LIN {X 0,Y 262.981,Z 430.812,A -85,B 0,C 180,E1 -18278.581,E2 -18278.581} C_VEL
LIN {X 0,Y 263.836,Z 425.981,A -85,B 0,C 180,E1 -18280.746,E2 -18280.746} C_VEL
LIN {X 0,Y 264.818,Z 420.507,A -85,B 0,C 180,E1 -18282.646,E2 -18282.646} C_VEL
LIN {X 0,Y 266.141,Z 413.615,A -85,B 0,C 180,E1 -18284.528,E2 -18284.528} C_VEL
LIN {X 0,Y 267.438,Z 405.7,A -85,B 0,C 180,E1 -18286.212,E2 -18286.212} C_VEL
LIN {X 0,Y 268.494,Z 398.154,A -85,B 0,C 180,E1 -18287.518,E2 -18287.518} C_VEL
LIN {X 0,Y 269.51,Z 390.236,A -85,B 0,C 180,E1 -18288.628,E2 -18288.628} C_VEL
LIN {X 0,Y 270.479,Z 382.045,A -85,B 0,C 180,E1 -18289.544,E2 -18289.544} C_VEL
LIN {X 0,Y 271.262,Z 373.736,A -85,B 0,C 180,E1 -18290.274,E2 -18290.274} C_VEL
LIN {X 0,Y 271.665,Z 364.754,A -85,B 0,C 180,E1 -18290.886,E2 -18290.886} C_VEL
LIN {X 0,Y 272.024,Z 355.186,A -85,B 0,C 180,E1 -18291.32,E2 -18291.32} C_VEL
LIN {X 0,Y 273.127,Z 306.683,A -85,B 0,C 180,E1 -18292.613,E2 -18292.613} C_VEL
LIN {X 0,Y 268.619,Z 295.095,A -85,B 0,C 180,E1 -18293.353,E2 -18293.353} C_VEL
LIN {X 0,Y 263.217,Z 282.947,A -85,B 0,C 180,E1 -18294.227,E2 -18294.227} C_VEL
LIN {X 0,Y 263.154,Z 282.519,A -85,B 0,C 180,E1 -18294.298,E2 -18294.298} C_VEL
LIN {X 0,Y 263.116,Z 282.525,A -85,B 0,C 180,E1 -18298.736,E2 -18298.736} C_VEL
LIN {X 0,Y 263.124,Z 282.523,A -85,B 0,C 180,E1 -18302.288,E2 -18302.288} C_VEL
LIN {X 0,Y 263.151,Z 282.514,A -85,B 0,C 180,E1 -18305.983,E2 -18305.983} C_VEL
LIN {X 0,Y 263.069,Z 282.528,A -85,B 0,C 180,E1 -18309.878,E2 -18309.878} C_VEL
LIN {X 0,Y 263.073,Z 282.528,A -85,B 0,C 180,E1 -18313.993,E2 -18313.993} C_VEL
LIN {X 0,Y 263.071,Z 282.519,A -85,B 0,C 180,E1 -18318.096,E2 -18318.096} C_VEL
LIN {X 0,Y 263.099,Z 282.522,A -85,B 0,C 180,E1 -18322.093,E2 -18322.093} C_VEL
LIN {X 0,Y 263.148,Z 282.518,A -85,B 0,C 180,E1 -18325.885,E2 -18325.885} C_VEL
LIN {X 0,Y 263.106,Z 282.524,A -85,B 0,C 180,E1 -18329.501,E2 -18329.501} C_VEL
LIN {X 0,Y 263.125,Z 282.517,A -85,B 0,C 180,E1 -18332.995,E2 -18332.995} C_VEL
LIN {X 0,Y 263.139,Z 282.517,A -85,B 0,C 180,E1 -18336.383,E2 -18336.383} C_VEL
LIN {X 0,Y 263.204,Z 282.511,A -85,B 0,C 180,E1 -18339.688,E2 -18339.688} C_VEL
LIN {X 0,Y 263.283,Z 282.49,A -85,B 0,C 180,E1 -18344.518,E2 -18344.518} C_VEL
LIN {X 0,Y 263.327,Z 282.496,A -85,B 0,C 180,E1 -18349.232,E2 -18349.232} C_VEL
LIN {X 0,Y 263.521,Z 282.471,A -85,B 0,C 180,E1 -18352.337,E2 -18352.337} C_VEL
LIN {X 0,Y 263.728,Z 282.438,A -85,B 0,C 180,E1 -18358.473,E2 -18358.473} C_VEL
LIN {X 0,Y 263.728,Z 282.444,A -85,B 0,C 180,E1 -18361.527,E2 -18361.527} C_VEL
LIN {X 0,Y 263.51,Z 282.471,A -85,B 0,C 180,E1 -18363.027,E2 -18363.027} C_VEL
LIN {X 0,Y 262.791,Z 282.568,A -85,B 0,C 180,E1 -18364.302,E2 -18364.302} C_VEL
LIN {X 0,Y 259.971,Z 282.922,A -85,B 0,C 180,E1 -18366.382,E2 -18366.382} C_VEL
LIN {X 0,Y 256.734,Z 283.316,A -85,B 0,C 180,E1 -18368.941,E2 -18368.941} C_VEL
LIN {X 0,Y 256.351,Z 283.36,A -85,B 0,C 180,E1 -18369.826,E2 -18369.826} C_VEL
LIN {X 0,Y 256.196,Z 283.384,A -85,B 0,C 180,E1 -18374.293,E2 -18374.293} C_VEL
LIN {X 0,Y 256.142,Z 283.39,A -85,B 0,C 180,E1 -18377.567,E2 -18377.567} C_VEL
LIN {X 0,Y 256.114,Z 283.392,A -85,B 0,C 180,E1 -18381.097,E2 -18381.097} C_VEL
LIN {X 0,Y 256.077,Z 283.396,A -85,B 0,C 180,E1 -18385.087,E2 -18385.087} C_VEL
LIN {X 0,Y 256.071,Z 283.4,A -85,B 0,C 180,E1 -18388.57,E2 -18388.57} C_VEL
LIN {X 0,Y 256.065,Z 283.404,A -85,B 0,C 180,E1 -18391.7,E2 -18391.7} C_VEL
LIN {X 0,Y 256.074,Z 283.402,A -85,B 0,C 180,E1 -18395.194,E2 -18395.194} C_VEL
LIN {X 0,Y 256.041,Z 283.407,A -85,B 0,C 180,E1 -18399.147,E2 -18399.147} C_VEL
LIN {X 0,Y 256.018,Z 283.41,A -85,B 0,C 180,E1 -18403.336,E2 -18403.336} C_VEL
LIN {X 0,Y 256.029,Z 283.405,A -85,B 0,C 180,E1 -18407.829,E2 -18407.829} C_VEL
LIN {X 0,Y 256.063,Z 283.403,A -85,B 0,C 180,E1 -18410.858,E2 -18410.858} C_VEL
LIN {X 0,Y 256.122,Z 283.395,A -85,B 0,C 180,E1 -18412.867,E2 -18412.867} C_VEL
LIN {X 0,Y 256.173,Z 283.581,A -85,B 0,C 180,E1 -18416.931,E2 -18416.931} C_VEL
LIN {X 0,Y 258.108,Z 292.95,A -85,B 0,C 180,E1 -18420.653,E2 -18420.653} C_VEL
LIN {X 0,Y 259.582,Z 301.431,A -85,B 0,C 180,E1 -18423.857,E2 -18423.857} C_VEL
LIN {X 0,Y 259.06,Z 305.592,A -85,B 0,C 180,E1 -18425.289,E2 -18425.289} C_VEL
LIN {X 0,Y 262.798,Z 329.088,A -85,B 0,C 180,E1 -18426.351,E2 -18426.351} C_VEL
LIN {X 0,Y 265.475,Z 352.015,A -85,B 0,C 180,E1 -18427.258,E2 -18427.258} C_VEL
LIN {X 0,Y 264.769,Z 384.627,A -85,B 0,C 180,E1 -18428.186,E2 -18428.186} C_VEL
LIN {X 0,Y 263.962,Z 395.927,A -85,B 0,C 180,E1 -18428.742,E2 -18428.742} C_VEL
LIN {X 0,Y 262.729,Z 407.426,A -85,B 0,C 180,E1 -18429.651,E2 -18429.651} C_VEL
LIN {X 0,Y 261.591,Z 416.12,A -85,B 0,C 180,E1 -18430.582,E2 -18430.582} C_VEL
LIN {X 0,Y 260.318,Z 424.431,A -85,B 0,C 180,E1 -18431.71,E2 -18431.71} C_VEL
LIN {X 0,Y 259.057,Z 432.309,A -85,B 0,C 180,E1 -18433.045,E2 -18433.045} C_VEL
LIN {X 0,Y 257.772,Z 439.681,A -85,B 0,C 180,E1 -18434.585,E2 -18434.585} C_VEL
LIN {X 0,Y 256.42,Z 447.167,A -85,B 0,C 180,E1 -18436.529,E2 -18436.529} C_VEL
LIN {X 0,Y 255.25,Z 454.012,A -85,B 0,C 180,E1 -18438.888,E2 -18438.888} C_VEL
LIN {X 0,Y 254.567,Z 459.229,A -85,B 0,C 180,E1 -18441.267,E2 -18441.267} C_VEL
LIN {X 0,Y 254.177,Z 463.065,A -85,B 0,C 180,E1 -18443.651,E2 -18443.651} C_VEL
LIN {X 0,Y 254.081,Z 464.833,A -85,B 0,C 180,E1 -18445.241,E2 -18445.241} C_VEL
LIN {X 0,Y 254.147,Z 466.105,A -85,B 0,C 180,E1 -18446.83,E2 -18446.83} C_VEL
LIN {X 0,Y 254.188,Z 466.894,A -85,B 0,C 180,E1 -18448.416,E2 -18448.416} C_VEL
LIN {X 0,Y 254.272,Z 467.194,A -85,B 0,C 180,E1 -18450.001,E2 -18450.001} C_VEL
LIN {X 0,Y 254.188,Z 466.886,A -85,B 0,C 180,E1 -18451.585,E2 -18451.585} C_VEL
LIN {X 0,Y 254.148,Z 466.082,A -85,B 0,C 180,E1 -18453.171,E2 -18453.171} C_VEL
LIN {X 0,Y 254.159,Z 464.076,A -85,B 0,C 180,E1 -18455.456,E2 -18455.456} C_VEL
LIN {X 0,Y 254.389,Z 460.655,A -85,B 0,C 180,E1 -18457.941,E2 -18457.941} C_VEL
LIN {X 0,Y 254.981,Z 455.856,A -85,B 0,C 180,E1 -18460.322,E2 -18460.322} C_VEL
LIN {X 0,Y 255.815,Z 450.672,A -85,B 0,C 180,E1 -18462.294,E2 -18462.294} C_VEL
LIN {X 0,Y 256.654,Z 445.61,A -85,B 0,C 180,E1 -18463.864,E2 -18463.864} C_VEL
LIN {X 0,Y 257.74,Z 439.523,A -85,B 0,C 180,E1 -18465.419,E2 -18465.419} C_VEL
LIN {X 0,Y 259.06,Z 432.125,A -85,B 0,C 180,E1 -18466.957,E2 -18466.957} C_VEL
LIN {X 0,Y 260.36,Z 424.206,A -85,B 0,C 180,E1 -18468.289,E2 -18468.289} C_VEL
LIN {X 0,Y 261.578,Z 415.838,A -85,B 0,C 180,E1 -18469.421,E2 -18469.421} C_VEL
LIN {X 0,Y 263.007,Z 404.764,A -85,B 0,C 180,E1 -18470.568,E2 -18470.568} C_VEL
LIN {X 0,Y 264.001,Z 394.383,A -85,B 0,C 180,E1 -18471.314,E2 -18471.314} C_VEL
LIN {X 0,Y 264.739,Z 384.752,A -85,B 0,C 180,E1 -18471.775,E2 -18471.775} C_VEL
LIN {X 0,Y 265.445,Z 352.252,A -85,B 0,C 180,E1 -18472.7,E2 -18472.7} C_VEL
LIN {X 0,Y 262.541,Z 327.679,A -85,B 0,C 180,E1 -18473.675,E2 -18473.675} C_VEL
LIN {X 0,Y 259.343,Z 307.499,A -85,B 0,C 180,E1 -18474.578,E2 -18474.578} C_VEL
LIN {X 0,Y 259.035,Z 305.586,A -85,B 0,C 180,E1 -18474.676,E2 -18474.676} C_VEL
LIN {X 0,Y 259.551,Z 301.335,A -85,B 0,C 180,E1 -18476.141,E2 -18476.141} C_VEL
LIN {X 0,Y 258.078,Z 292.765,A -85,B 0,C 180,E1 -18479.376,E2 -18479.376} C_VEL
LIN {X 0,Y 256.134,Z 283.389,A -85,B 0,C 180,E1 -18483.141,E2 -18483.141} C_VEL
LIN {X 0,Y 256.111,Z 283.397,A -85,B 0,C 180,E1 -18487.27,E2 -18487.27} C_VEL
LIN {X 0,Y 256.019,Z 283.409,A -85,B 0,C 180,E1 -18491.211,E2 -18491.211} C_VEL
LIN {X 0,Y 256.018,Z 283.407,A -85,B 0,C 180,E1 -18495.54,E2 -18495.54} C_VEL
LIN {X 0,Y 256.01,Z 283.411,A -85,B 0,C 180,E1 -18498.788,E2 -18498.788} C_VEL
LIN {X 0,Y 256.1,Z 283.399,A -85,B 0,C 180,E1 -18502.862,E2 -18502.862} C_VEL
LIN {X 0,Y 256.067,Z 283.402,A -85,B 0,C 180,E1 -18506.707,E2 -18506.707} C_VEL
LIN {X 0,Y 256.042,Z 283.406,A -85,B 0,C 180,E1 -18510.391,E2 -18510.391} C_VEL
LIN {X 0,Y 256.067,Z 283.402,A -85,B 0,C 180,E1 -18513.951,E2 -18513.951} C_VEL
LIN {X 0,Y 256.058,Z 283.401,A -85,B 0,C 180,E1 -18517.403,E2 -18517.403} C_VEL
LIN {X 0,Y 256.101,Z 283.395,A -85,B 0,C 180,E1 -18520.773,E2 -18520.773} C_VEL
LIN {X 0,Y 256.214,Z 283.382,A -85,B 0,C 180,E1 -18524.08,E2 -18524.08} C_VEL
LIN {X 0,Y 256.272,Z 283.37,A -85,B 0,C 180,E1 -18528.933,E2 -18528.933} C_VEL
LIN {X 0,Y 256.458,Z 283.334,A -85,B 0,C 180,E1 -18532.125,E2 -18532.125} C_VEL
LIN {X 0,Y 256.445,Z 283.351,A -85,B 0,C 180,E1 -18536.858,E2 -18536.858} C_VEL
LIN {X 0,Y 256.695,Z 283.32,A -85,B 0,C 180,E1 -18538.431,E2 -18538.431} C_VEL
LIN {X 0,Y 256.697,Z 283.312,A -85,B 0,C 180,E1 -18541.569,E2 -18541.569} C_VEL
LIN {X 0,Y 256.444,Z 283.345,A -85,B 0,C 180,E1 -18546.573,E2 -18546.573} C_VEL
LIN {X 0,Y 256.405,Z 283.359,A -85,B 0,C 180,E1 -18549.466,E2 -18549.466} C_VEL
LIN {X 0,Y 256.208,Z 283.369,A -85,B 0,C 180,E1 -18554.293,E2 -18554.293} C_VEL
LIN {X 0,Y 256.149,Z 283.385,A -85,B 0,C 180,E1 -18557.566,E2 -18557.566} C_VEL
LIN {X 0,Y 256.121,Z 283.393,A -85,B 0,C 180,E1 -18561.097,E2 -18561.097} C_VEL
LIN {X 0,Y 256.085,Z 283.398,A -85,B 0,C 180,E1 -18565.087,E2 -18565.087} C_VEL
LIN {X 0,Y 256.079,Z 283.397,A -85,B 0,C 180,E1 -18568.57,E2 -18568.57} C_VEL
LIN {X 0,Y 256.072,Z 283.397,A -85,B 0,C 180,E1 -18571.699,E2 -18571.699} C_VEL
LIN {X 0,Y 256.08,Z 283.388,A -85,B 0,C 180,E1 -18575.193,E2 -18575.193} C_VEL
LIN {X 0,Y 256.044,Z 283.403,A -85,B 0,C 180,E1 -18579.147,E2 -18579.147} C_VEL
LIN {X 0,Y 256.023,Z 283.399,A -85,B 0,C 180,E1 -18583.335,E2 -18583.335} C_VEL
LIN {X 0,Y 256.036,Z 283.404,A -85,B 0,C 180,E1 -18587.828,E2 -18587.828} C_VEL
LIN {X 0,Y 256.067,Z 283.378,A -85,B 0,C 180,E1 -18590.856,E2 -18590.856} C_VEL
LIN {X 0,Y 256.081,Z 283.395,A -85,B 0,C 180,E1 -18594.806,E2 -18594.806} C_VEL
LIN {X 0,Y 256.079,Z 283.398,A -85,B 0,C 180,E1 -18598.57,E2 -18598.57} C_VEL
LIN {X 0,Y 256.081,Z 283.399,A -85,B 0,C 180,E1 -18602.188,E2 -18602.188} C_VEL
LIN {X 0,Y 256.164,Z 283.505,A -85,B 0,C 180,E1 -18605.198,E2 -18605.198} C_VEL
LIN {X 0,Y 257.229,Z 286.37,A -85,B 0,C 180,E1 -18605.397,E2 -18605.397} C_VEL
LIN {X 0,Y 264.851,Z 303.493,A -85,B 0,C 180,E1 -18606.662,E2 -18606.662} C_VEL
LIN {X 0,Y 266.558,Z 308.226,A -85,B 0,C 180,E1 -18606.959,E2 -18606.959} C_VEL
LIN {X 0,Y 265.305,Z 356.614,A -85,B 0,C 180,E1 -18608.281,E2 -18608.281} C_VEL
LIN {X 0,Y 264.934,Z 366.352,A -85,B 0,C 180,E1 -18608.76,E2 -18608.76} C_VEL
LIN {X 0,Y 264.292,Z 377.392,A -85,B 0,C 180,E1 -18609.572,E2 -18609.572} C_VEL
LIN {X 0,Y 263.081,Z 388.176,A -85,B 0,C 180,E1 -18610.695,E2 -18610.695} C_VEL
LIN {X 0,Y 262.117,Z 395.319,A -85,B 0,C 180,E1 -18611.636,E2 -18611.636} C_VEL
LIN {X 0,Y 260.971,Z 403.419,A -85,B 0,C 180,E1 -18612.97,E2 -18612.97} C_VEL
LIN {X 0,Y 259.915,Z 410.098,A -85,B 0,C 180,E1 -18614.311,E2 -18614.311} C_VEL
LIN {X 0,Y 258.791,Z 416.422,A -85,B 0,C 180,E1 -18615.852,E2 -18615.852} C_VEL
LIN {X 0,Y 257.743,Z 421.68,A -85,B 0,C 180,E1 -18617.399,E2 -18617.399} C_VEL
LIN {X 0,Y 256.886,Z 426.065,A -85,B 0,C 180,E1 -18618.958,E2 -18618.958} C_VEL
LIN {X 0,Y 256.235,Z 429.71,A -85,B 0,C 180,E1 -18620.527,E2 -18620.527} C_VEL
LIN {X 0,Y 255.713,Z 432.686,A -85,B 0,C 180,E1 -18622.101,E2 -18622.101} C_VEL
LIN {X 0,Y 255.241,Z 434.992,A -85,B 0,C 180,E1 -18623.676,E2 -18623.676} C_VEL
LIN {X 0,Y 254.819,Z 436.748,A -85,B 0,C 180,E1 -18625.253,E2 -18625.253} C_VEL
LIN {X 0,Y 254.53,Z 438.013,A -85,B 0,C 180,E1 -18626.834,E2 -18626.834} C_VEL
LIN {X 0,Y 254.358,Z 438.81,A -85,B 0,C 180,E1 -18628.416,E2 -18628.416} C_VEL
LIN {X 0,Y 254.305,Z 439.113,A -85,B 0,C 180,E1 -18629.999,E2 -18629.999} C_VEL
LIN {X 0,Y 254.355,Z 438.836,A -85,B 0,C 180,E1 -18631.582,E2 -18631.582} C_VEL
LIN {X 0,Y 254.518,Z 438.09,A -85,B 0,C 180,E1 -18633.165,E2 -18633.165} C_VEL
LIN {X 0,Y 254.813,Z 436.878,A -85,B 0,C 180,E1 -18634.745,E2 -18634.745} C_VEL
LIN {X 0,Y 255.443,Z 434.037,A -85,B 0,C 180,E1 -18637.111,E2 -18637.111} C_VEL
LIN {X 0,Y 255.943,Z 431.454,A -85,B 0,C 180,E1 -18638.685,E2 -18638.685} C_VEL
LIN {X 0,Y 256.878,Z 426.37,A -85,B 0,C 180,E1 -18641.04,E2 -18641.04} C_VEL
LIN {X 0,Y 257.918,Z 420.896,A -85,B 0,C 180,E1 -18642.99,E2 -18642.99} C_VEL
LIN {X 0,Y 259.284,Z 414.003,A -85,B 0,C 180,E1 -18644.921,E2 -18644.921} C_VEL
LIN {X 0,Y 260.646,Z 406.088,A -85,B 0,C 180,E1 -18646.647,E2 -18646.647} C_VEL
LIN {X 0,Y 261.751,Z 398.541,A -85,B 0,C 180,E1 -18647.984,E2 -18647.984} C_VEL
LIN {X 0,Y 262.817,Z 390.621,A -85,B 0,C 180,E1 -18649.121,E2 -18649.121} C_VEL
LIN {X 0,Y 263.835,Z 382.429,A -85,B 0,C 180,E1 -18650.057,E2 -18650.057} C_VEL
LIN {X 0,Y 264.639,Z 374.119,A -85,B 0,C 180,E1 -18650.805,E2 -18650.805} C_VEL
LIN {X 0,Y 265.066,Z 365.134,A -85,B 0,C 180,E1 -18651.431,E2 -18651.431} C_VEL
LIN {X 0,Y 265.444,Z 355.6,A -85,B 0,C 180,E1 -18651.874,E2 -18651.874} C_VEL
LIN {X 0,Y 266.661,Z 308.565,A -85,B 0,C 180,E1 -18653.15,E2 -18653.15} C_VEL
LIN {X 0,Y 262.754,Z 298.437,A -85,B 0,C 180,E1 -18653.818,E2 -18653.818} C_VEL
LIN {X 0,Y 256.205,Z 284.082,A -85,B 0,C 180,E1 -18654.912,E2 -18654.912} C_VEL
LIN {X 0,Y 256.092,Z 283.403,A -85,B 0,C 180,E1 -18654.995,E2 -18654.995} C_VEL
LIN {X 0,Y 256.074,Z 283.402,A -85,B 0,C 180,E1 -18658.568,E2 -18658.568} C_VEL
LIN {X 0,Y 256.068,Z 283.4,A -85,B 0,C 180,E1 -18661.698,E2 -18661.698} C_VEL
LIN {X 0,Y 256.076,Z 283.396,A -85,B 0,C 180,E1 -18665.193,E2 -18665.193} C_VEL
LIN {X 0,Y 256.039,Z 283.403,A -85,B 0,C 180,E1 -18669.147,E2 -18669.147} C_VEL
LIN {X 0,Y 256.018,Z 283.403,A -85,B 0,C 180,E1 -18673.335,E2 -18673.335} C_VEL
LIN {X 0,Y 256.026,Z 283.395,A -85,B 0,C 180,E1 -18677.829,E2 -18677.829} C_VEL
LIN {X 0,Y 256.038,Z 283.4,A -85,B 0,C 180,E1 -18680.852,E2 -18680.852} C_VEL
LIN {X 0,Y 256.074,Z 283.396,A -85,B 0,C 180,E1 -18684.806,E2 -18684.806} C_VEL
LIN {X 0,Y 256.074,Z 283.396,A -85,B 0,C 180,E1 -18688.57,E2 -18688.57} C_VEL
LIN {X 0,Y 256.082,Z 283.393,A -85,B 0,C 180,E1 -18692.189,E2 -18692.189} C_VEL
LIN {X 0,Y 256.128,Z 283.392,A -85,B 0,C 180,E1 -18695.695,E2 -18695.695} C_VEL
LIN {X 0,Y 256.119,Z 283.394,A -85,B 0,C 180,E1 -18699.101,E2 -18699.101} C_VEL
LIN {X 0,Y 256.208,Z 283.37,A -85,B 0,C 180,E1 -18704.079,E2 -18704.079} C_VEL
LIN {X 0,Y 256.271,Z 283.374,A -85,B 0,C 180,E1 -18708.932,E2 -18708.932} C_VEL
LIN {X 0,Y 256.463,Z 283.349,A -85,B 0,C 180,E1 -18712.125,E2 -18712.125} C_VEL
LIN {X 0,Y 256.443,Z 283.338,A -85,B 0,C 180,E1 -18716.858,E2 -18716.858} C_VEL
LIN {X 0,Y 256.69,Z 283.313,A -85,B 0,C 180,E1 -18718.431,E2 -18718.431} C_VEL
LIN {X 0,Y 256.69,Z 283.321,A -85,B 0,C 180,E1 -18721.569,E2 -18721.569} C_VEL
LIN {X 0,Y 256.448,Z 283.352,A -85,B 0,C 180,E1 -18726.293,E2 -18726.293} C_VEL
LIN {X 0,Y 256.397,Z 283.356,A -85,B 0,C 180,E1 -18729.466,E2 -18729.466} C_VEL
LIN {X 0,Y 256.351,Z 283.36,A -85,B 0,C 180,E1 -18729.826,E2 -18729.826} C_VEL
LIN {X 0,Y 255.59,Z 283.457,A -85,B 0,C 180,E1 -18731.135,E2 -18731.135} C_VEL
LIN {X 0,Y 252.714,Z 283.817,A -85,B 0,C 180,E1 -18733.27,E2 -18733.27} C_VEL
LIN {X 0,Y 250.299,Z 284.12,A -85,B 0,C 180,E1 -18735.006,E2 -18735.006} C_VEL
LIN {X 0,Y 249.225,Z 284.253,A -85,B 0,C 180,E1 -18736.352,E2 -18736.352} C_VEL
LIN {X 0,Y 249.113,Z 284.265,A -85,B 0,C 180,E1 -18736.809,E2 -18736.809} C_VEL
LIN {X 0,Y 249.038,Z 284.275,A -85,B 0,C 180,E1 -18741.522,E2 -18741.522} C_VEL
LIN {X 0,Y 249.038,Z 284.275,A -85,B 0,C 180,E1 -18745.44,E2 -18745.44} C_VEL
LIN {X 0,Y 249.019,Z 284.279,A -85,B 0,C 180,E1 -18748.968,E2 -18748.968} C_VEL
LIN {X 0,Y 249.021,Z 284.279,A -85,B 0,C 180,E1 -18752.427,E2 -18752.427} C_VEL
LIN {X 0,Y 249.006,Z 284.281,A -85,B 0,C 180,E1 -18756.349,E2 -18756.349} C_VEL
LIN {X 0,Y 248.971,Z 284.285,A -85,B 0,C 180,E1 -18760.485,E2 -18760.485} C_VEL
LIN {X 0,Y 248.958,Z 284.289,A -85,B 0,C 180,E1 -18764.889,E2 -18764.889} C_VEL
LIN {X 0,Y 248.975,Z 284.287,A -85,B 0,C 180,E1 -18767.355,E2 -18767.355} C_VEL
LIN {X 0,Y 249.037,Z 284.276,A -85,B 0,C 180,E1 -18772.202,E2 -18772.202} C_VEL
LIN {X 0,Y 249.076,Z 284.43,A -85,B 0,C 180,E1 -18776.378,E2 -18776.378} C_VEL
LIN {X 0,Y 251.064,Z 293.716,A -85,B 0,C 180,E1 -18780.201,E2 -18780.201} C_VEL
LIN {X 0,Y 252.606,Z 302.339,A -85,B 0,C 180,E1 -18783.568,E2 -18783.568} C_VEL
LIN {X 0,Y 252.335,Z 305.187,A -85,B 0,C 180,E1 -18784.586,E2 -18784.586} C_VEL
LIN {X 0,Y 256.291,Z 330.056,A -85,B 0,C 180,E1 -18785.753,E2 -18785.753} C_VEL
LIN {X 0,Y 258.774,Z 351.122,A -85,B 0,C 180,E1 -18786.62,E2 -18786.62} C_VEL
LIN {X 0,Y 258.889,Z 358.477,A -85,B 0,C 180,E1 -18786.847,E2 -18786.847} C_VEL
LIN {X 0,Y 258.164,Z 384.249,A -85,B 0,C 180,E1 -18787.598,E2 -18787.598} C_VEL
LIN {X 0,Y 257.321,Z 396.001,A -85,B 0,C 180,E1 -18788.198,E2 -18788.198} C_VEL
LIN {X 0,Y 256.091,Z 407.04,A -85,B 0,C 180,E1 -18789.099,E2 -18789.099} C_VEL
LIN {X 0,Y 254.911,Z 415.733,A -85,B 0,C 180,E1 -18790.052,E2 -18790.052} C_VEL
LIN {X 0,Y 253.575,Z 424.042,A -85,B 0,C 180,E1 -18791.205,E2 -18791.205} C_VEL
LIN {X 0,Y 252.252,Z 431.919,A -85,B 0,C 180,E1 -18792.573,E2 -18792.573} C_VEL
LIN {X 0,Y 250.896,Z 439.29,A -85,B 0,C 180,E1 -18794.151,E2 -18794.151} C_VEL
LIN {X 0,Y 249.505,Z 446.776,A -85,B 0,C 180,E1 -18796.148,E2 -18796.148} C_VEL
LIN {X 0,Y 248.261,Z 453.62,A -85,B 0,C 180,E1 -18798.571,E2 -18798.571} C_VEL
LIN {X 0,Y 247.528,Z 458.837,A -85,B 0,C 180,E1 -18801.017,E2 -18801.017} C_VEL
LIN {X 0,Y 247.095,Z 462.673,A -85,B 0,C 180,E1 -18803.468,E2 -18803.468} C_VEL
LIN {X 0,Y 247.009,Z 464.442,A -85,B 0,C 180,E1 -18805.104,E2 -18805.104} C_VEL
LIN {X 0,Y 247.056,Z 465.713,A -85,B 0,C 180,E1 -18806.739,E2 -18806.739} C_VEL
LIN {X 0,Y 247.112,Z 466.503,A -85,B 0,C 180,E1 -18808.371,E2 -18808.371} C_VEL
LIN {X 0,Y 247.191,Z 466.803,A -85,B 0,C 180,E1 -18810.001,E2 -18810.001} C_VEL
LIN {X 0,Y 247.112,Z 466.495,A -85,B 0,C 180,E1 -18811.631,E2 -18811.631} C_VEL
LIN {X 0,Y 247.058,Z 465.69,A -85,B 0,C 180,E1 -18813.262,E2 -18813.262} C_VEL
LIN {X 0,Y 247.048,Z 463.966,A -85,B 0,C 180,E1 -18815.332,E2 -18815.332} C_VEL
LIN {X 0,Y 247.199,Z 461.449,A -85,B 0,C 180,E1 -18817.351,E2 -18817.351} C_VEL
LIN {X 0,Y 247.528,Z 458.765,A -85,B 0,C 180,E1 -18818.985,E2 -18818.985} C_VEL
LIN {X 0,Y 248.261,Z 453.526,A -85,B 0,C 180,E1 -18821.43,E2 -18821.43} C_VEL
LIN {X 0,Y 249.501,Z 446.639,A -85,B 0,C 180,E1 -18823.854,E2 -18823.854} C_VEL
LIN {X 0,Y 250.874,Z 439.127,A -85,B 0,C 180,E1 -18825.852,E2 -18825.852} C_VEL
LIN {X 0,Y 252.256,Z 431.729,A -85,B 0,C 180,E1 -18827.428,E2 -18827.428} C_VEL
LIN {X 0,Y 253.625,Z 423.81,A -85,B 0,C 180,E1 -18828.793,E2 -18828.793} C_VEL
LIN {X 0,Y 254.897,Z 415.441,A -85,B 0,C 180,E1 -18829.951,E2 -18829.951} C_VEL
LIN {X 0,Y 256.378,Z 404.365,A -85,B 0,C 180,E1 -18831.125,E2 -18831.125} C_VEL
LIN {X 0,Y 257.451,Z 393.688,A -85,B 0,C 180,E1 -18831.902,E2 -18831.902} C_VEL
LIN {X 0,Y 258.141,Z 384.504,A -85,B 0,C 180,E1 -18832.355,E2 -18832.355} C_VEL
LIN {X 0,Y 258.876,Z 352.874,A -85,B 0,C 180,E1 -18833.279,E2 -18833.279} C_VEL
LIN {X 0,Y 256.108,Z 329.071,A -85,B 0,C 180,E1 -18834.254,E2 -18834.254} C_VEL
LIN {X 0,Y 252.722,Z 307.666,A -85,B 0,C 180,E1 -18835.248,E2 -18835.248} C_VEL
LIN {X 0,Y 252.309,Z 305.175,A -85,B 0,C 180,E1 -18835.38,E2 -18835.38} C_VEL
LIN {X 0,Y 252.582,Z 302.221,A -85,B 0,C 180,E1 -18836.437,E2 -18836.437} C_VEL
LIN {X 0,Y 250.837,Z 292.374,A -85,B 0,C 180,E1 -18840.288,E2 -18840.288} C_VEL
LIN {X 0,Y 249.058,Z 284.27,A -85,B 0,C 180,E1 -18843.688,E2 -18843.688} C_VEL
LIN {X 0,Y 249.023,Z 284.278,A -85,B 0,C 180,E1 -18848.382,E2 -18848.382} C_VEL
LIN {X 0,Y 248.971,Z 284.287,A -85,B 0,C 180,E1 -18852.783,E2 -18852.783} C_VEL
LIN {X 0,Y 248.978,Z 284.285,A -85,B 0,C 180,E1 -18857.355,E2 -18857.355} C_VEL
LIN {X 0,Y 249.022,Z 284.28,A -85,B 0,C 180,E1 -18862.208,E2 -18862.208} C_VEL
LIN {X 0,Y 249.044,Z 284.275,A -85,B 0,C 180,E1 -18865.64,E2 -18865.64} C_VEL
LIN {X 0,Y 248.995,Z 284.281,A -85,B 0,C 180,E1 -18869.466,E2 -18869.466} C_VEL
LIN {X 0,Y 249.014,Z 284.278,A -85,B 0,C 180,E1 -18873.156,E2 -18873.156} C_VEL
LIN {X 0,Y 249.007,Z 284.28,A -85,B 0,C 180,E1 -18876.726,E2 -18876.726} C_VEL
LIN {X 0,Y 249.04,Z 284.276,A -85,B 0,C 180,E1 -18880.206,E2 -18880.206} C_VEL
LIN {X 0,Y 249.16,Z 284.261,A -85,B 0,C 180,E1 -18883.617,E2 -18883.617} C_VEL
LIN {X 0,Y 249.217,Z 284.249,A -85,B 0,C 180,E1 -18888.615,E2 -18888.615} C_VEL
LIN {X 0,Y 249.405,Z 284.211,A -85,B 0,C 180,E1 -18891.901,E2 -18891.901} C_VEL
LIN {X 0,Y 249.256,Z 284.242,A -85,B 0,C 180,E1 -18895.148,E2 -18895.148} C_VEL
LIN {X 0,Y 249.656,Z 284.197,A -85,B 0,C 180,E1 -18898.387,E2 -18898.387} C_VEL
LIN {X 0,Y 249.658,Z 284.187,A -85,B 0,C 180,E1 -18901.613,E2 -18901.613} C_VEL
LIN {X 0,Y 249.422,Z 284.22,A -85,B 0,C 180,E1 -18906.55,E2 -18906.55} C_VEL
LIN {X 0,Y 249.335,Z 284.238,A -85,B 0,C 180,E1 -18909.737,E2 -18909.737} C_VEL
LIN {X 0,Y 249.151,Z 284.245,A -85,B 0,C 180,E1 -18914.707,E2 -18914.707} C_VEL
LIN {X 0,Y 249.081,Z 284.265,A -85,B 0,C 180,E1 -18918.082,E2 -18918.082} C_VEL
LIN {X 0,Y 249.045,Z 284.273,A -85,B 0,C 180,E1 -18921.522,E2 -18921.522} C_VEL
LIN {X 0,Y 249.046,Z 284.274,A -85,B 0,C 180,E1 -18925.439,E2 -18925.439} C_VEL
LIN {X 0,Y 249.027,Z 284.277,A -85,B 0,C 180,E1 -18928.968,E2 -18928.968} C_VEL
LIN {X 0,Y 249.028,Z 284.274,A -85,B 0,C 180,E1 -18932.426,E2 -18932.426} C_VEL
LIN {X 0,Y 249.013,Z 284.272,A -85,B 0,C 180,E1 -18936.349,E2 -18936.349} C_VEL
LIN {X 0,Y 248.974,Z 284.282,A -85,B 0,C 180,E1 -18940.485,E2 -18940.485} C_VEL
LIN {X 0,Y 248.964,Z 284.286,A -85,B 0,C 180,E1 -18944.888,E2 -18944.888} C_VEL
LIN {X 0,Y 248.981,Z 284.284,A -85,B 0,C 180,E1 -18947.355,E2 -18947.355} C_VEL
LIN {X 0,Y 249.045,Z 284.247,A -85,B 0,C 180,E1 -18952.2,E2 -18952.2} C_VEL
LIN {X 0,Y 249.045,Z 284.274,A -85,B 0,C 180,E1 -18955.639,E2 -18955.639} C_VEL
LIN {X 0,Y 248.996,Z 284.282,A -85,B 0,C 180,E1 -18959.465,E2 -18959.465} C_VEL
LIN {X 0,Y 249.025,Z 284.28,A -85,B 0,C 180,E1 -18963.156,E2 -18963.156} C_VEL
LIN {X 0,Y 249.096,Z 284.45,A -85,B 0,C 180,E1 -18964.46,E2 -18964.46} C_VEL
LIN {X 0,Y 250.147,Z 287.197,A -85,B 0,C 180,E1 -18964.663,E2 -18964.663} C_VEL
LIN {X 0,Y 258.118,Z 304.653,A -85,B 0,C 180,E1 -18966.037,E2 -18966.037} C_VEL
LIN {X 0,Y 260.08,Z 310.304,A -85,B 0,C 180,E1 -18966.4,E2 -18966.4} C_VEL
LIN {X 0,Y 258.783,Z 355.728,A -85,B 0,C 180,E1 -18967.653,E2 -18967.653} C_VEL
LIN {X 0,Y 258.446,Z 365.095,A -85,B 0,C 180,E1 -18968.095,E2 -18968.095} C_VEL
LIN {X 0,Y 257.918,Z 374.201,A -85,B 0,C 180,E1 -18968.73,E2 -18968.73} C_VEL
LIN {X 0,Y 257.038,Z 383.51,A -85,B 0,C 180,E1 -18969.597,E2 -18969.597} C_VEL
LIN {X 0,Y 255.718,Z 393.062,A -85,B 0,C 180,E1 -18970.743,E2 -18970.743} C_VEL
LIN {X 0,Y 254.369,Z 402.799,A -85,B 0,C 180,E1 -18972.306,E2 -18972.306} C_VEL
LIN {X 0,Y 253.104,Z 410.492,A -85,B 0,C 180,E1 -18973.878,E2 -18973.878} C_VEL
LIN {X 0,Y 251.916,Z 416.817,A -85,B 0,C 180,E1 -18975.458,E2 -18975.458} C_VEL
LIN {X 0,Y 250.846,Z 422.073,A -85,B 0,C 180,E1 -18977.047,E2 -18977.047} C_VEL
LIN {X 0,Y 249.936,Z 426.458,A -85,B 0,C 180,E1 -18978.647,E2 -18978.647} C_VEL
LIN {X 0,Y 249.237,Z 430.103,A -85,B 0,C 180,E1 -18980.259,E2 -18980.259} C_VEL
LIN {X 0,Y 248.682,Z 433.079,A -85,B 0,C 180,E1 -18981.876,E2 -18981.876} C_VEL
LIN {X 0,Y 248.22,Z 435.383,A -85,B 0,C 180,E1 -18983.496,E2 -18983.496} C_VEL
LIN {X 0,Y 247.774,Z 437.14,A -85,B 0,C 180,E1 -18985.118,E2 -18985.118} C_VEL
LIN {X 0,Y 247.466,Z 438.404,A -85,B 0,C 180,E1 -18986.743,E2 -18986.743} C_VEL
LIN {X 0,Y 247.282,Z 439.201,A -85,B 0,C 180,E1 -18988.371,E2 -18988.371} C_VEL
LIN {X 0,Y 247.225,Z 439.504,A -85,B 0,C 180,E1 -18989.999,E2 -18989.999} C_VEL
LIN {X 0,Y 247.278,Z 439.226,A -85,B 0,C 180,E1 -18991.628,E2 -18991.628} C_VEL
LIN {X 0,Y 247.454,Z 438.481,A -85,B 0,C 180,E1 -18993.255,E2 -18993.255} C_VEL
LIN {X 0,Y 247.768,Z 437.268,A -85,B 0,C 180,E1 -18994.881,E2 -18994.881} C_VEL
LIN {X 0,Y 248.418,Z 434.427,A -85,B 0,C 180,E1 -18997.313,E2 -18997.313} C_VEL
LIN {X 0,Y 248.877,Z 432.183,A -85,B 0,C 180,E1 -18998.749,E2 -18998.749} C_VEL
LIN {X 0,Y 249.926,Z 426.76,A -85,B 0,C 180,E1 -19001.351,E2 -19001.351} C_VEL
LIN {X 0,Y 251.03,Z 421.284,A -85,B 0,C 180,E1 -19003.353,E2 -19003.353} C_VEL
LIN {X 0,Y 252.441,Z 414.392,A -85,B 0,C 180,E1 -19005.335,E2 -19005.335} C_VEL
LIN {X 0,Y 253.874,Z 406.475,A -85,B 0,C 180,E1 -19007.105,E2 -19007.105} C_VEL
LIN {X 0,Y 255.031,Z 398.927,A -85,B 0,C 180,E1 -19008.475,E2 -19008.475} C_VEL
LIN {X 0,Y 256.152,Z 391.006,A -85,B 0,C 180,E1 -19009.639,E2 -19009.639} C_VEL
LIN {X 0,Y 257.21,Z 382.813,A -85,B 0,C 180,E1 -19010.596,E2 -19010.596} C_VEL
LIN {X 0,Y 258.037,Z 374.501,A -85,B 0,C 180,E1 -19011.363,E2 -19011.363} C_VEL
LIN {X 0,Y 258.499,Z 365.513,A -85,B 0,C 180,E1 -19012.004,E2 -19012.004} C_VEL
LIN {X 0,Y 258.875,Z 356.199,A -85,B 0,C 180,E1 -19012.45,E2 -19012.45} C_VEL
LIN {X 0,Y 260.077,Z 309.942,A -85,B 0,C 180,E1 -19013.741,E2 -19013.741} C_VEL
LIN {X 0,Y 255.636,Z 299.007,A -85,B 0,C 180,E1 -19014.519,E2 -19014.519} C_VEL
LIN {X 0,Y 249.148,Z 284.96,A -85,B 0,C 180,E1 -19015.653,E2 -19015.653} C_VEL
LIN {X 0,Y 249.023,Z 284.282,A -85,B 0,C 180,E1 -19015.757,E2 -19015.757} C_VEL
LIN {X 0,Y 249.022,Z 284.279,A -85,B 0,C 180,E1 -19018.967,E2 -19018.967} C_VEL
LIN {X 0,Y 249.024,Z 284.28,A -85,B 0,C 180,E1 -19022.426,E2 -19022.426} C_VEL
LIN {X 0,Y 249.008,Z 284.275,A -85,B 0,C 180,E1 -19026.348,E2 -19026.348} C_VEL
LIN {X 0,Y 248.969,Z 284.278,A -85,B 0,C 180,E1 -19030.484,E2 -19030.484} C_VEL
LIN {X 0,Y 248.959,Z 284.284,A -85,B 0,C 180,E1 -19034.888,E2 -19034.888} C_VEL
LIN {X 0,Y 248.973,Z 284.274,A -85,B 0,C 180,E1 -19037.353,E2 -19037.353} C_VEL
LIN {X 0,Y 249.017,Z 284.276,A -85,B 0,C 180,E1 -19042.206,E2 -19042.206} C_VEL
LIN {X 0,Y 249.039,Z 284.276,A -85,B 0,C 180,E1 -19045.638,E2 -19045.638} C_VEL
LIN {X 0,Y 248.991,Z 284.282,A -85,B 0,C 180,E1 -19049.465,E2 -19049.465} C_VEL
LIN {X 0,Y 249.026,Z 284.274,A -85,B 0,C 180,E1 -19053.156,E2 -19053.156} C_VEL
LIN {X 0,Y 249.047,Z 284.273,A -85,B 0,C 180,E1 -19056.729,E2 -19056.729} C_VEL
LIN {X 0,Y 249.04,Z 284.274,A -85,B 0,C 180,E1 -19060.205,E2 -19060.205} C_VEL
LIN {X 0,Y 249.153,Z 284.25,A -85,B 0,C 180,E1 -19063.616,E2 -19063.616} C_VEL
LIN {X 0,Y 249.216,Z 284.25,A -85,B 0,C 180,E1 -19068.615,E2 -19068.615} C_VEL
LIN {X 0,Y 249.409,Z 284.227,A -85,B 0,C 180,E1 -19071.9,E2 -19071.9} C_VEL
LIN {X 0,Y 249.253,Z 284.233,A -85,B 0,C 180,E1 -19075.147,E2 -19075.147} C_VEL
LIN {X 0,Y 249.651,Z 284.189,A -85,B 0,C 180,E1 -19078.387,E2 -19078.387} C_VEL
LIN {X 0,Y 249.651,Z 284.198,A -85,B 0,C 180,E1 -19081.613,E2 -19081.613} C_VEL
LIN {X 0,Y 249.422,Z 284.228,A -85,B 0,C 180,E1 -19086.471,E2 -19086.471} C_VEL
LIN {X 0,Y 249.322,Z 284.238,A -85,B 0,C 180,E1 -19089.779,E2 -19089.779} C_VEL
LIN {X 0,Y 249.141,Z 284.261,A -85,B 0,C 180,E1 -19094.707,E2 -19094.707} C_VEL
LIN {X 0,Y 249.113,Z 284.265,A -85,B 0,C 180,E1 -19096.809,E2 -19096.809} C_VEL
LIN {X 0,Y 248.386,Z 284.359,A -85,B 0,C 180,E1 -19098.158,E2 -19098.158} C_VEL
LIN {X 0,Y 245.538,Z 284.716,A -85,B 0,C 180,E1 -19100.358,E2 -19100.358} C_VEL
LIN {X 0,Y 243.136,Z 285.017,A -85,B 0,C 180,E1 -19102.149,E2 -19102.149} C_VEL
LIN {X 0,Y 242.078,Z 285.145,A -85,B 0,C 180,E1 -19103.538,E2 -19103.538} C_VEL
LIN {X 0,Y 241.975,Z 285.155,A -85,B 0,C 180,E1 -19104.008,E2 -19104.008} C_VEL
LIN {X 0,Y 241.946,Z 285.162,A -85,B 0,C 180,E1 -19107.695,E2 -19107.695} C_VEL
LIN {X 0,Y 241.944,Z 285.163,A -85,B 0,C 180,E1 -19111.524,E2 -19111.524} C_VEL
LIN {X 0,Y 241.974,Z 285.16,A -85,B 0,C 180,E1 -19115.588,E2 -19115.588} C_VEL
LIN {X 0,Y 241.928,Z 285.165,A -85,B 0,C 180,E1 -19119.724,E2 -19119.724} C_VEL
LIN {X 0,Y 241.892,Z 285.167,A -85,B 0,C 180,E1 -19124.211,E2 -19124.211} C_VEL
LIN {X 0,Y 241.904,Z 285.165,A -85,B 0,C 180,E1 -19128.072,E2 -19128.072} C_VEL
LIN {X 0,Y 241.98,Z 285.156,A -85,B 0,C 180,E1 -19132.418,E2 -19132.418} C_VEL
LIN {X 0,Y 242.041,Z 285.199,A -85,B 0,C 180,E1 -19135.767,E2 -19135.767} C_VEL
LIN {X 0,Y 244.146,Z 295.222,A -85,B 0,C 180,E1 -19140.026,E2 -19140.026} C_VEL
LIN {X 0,Y 245.636,Z 303.512,A -85,B 0,C 180,E1 -19143.362,E2 -19143.362} C_VEL
LIN {X 0,Y 245.626,Z 304.738,A -85,B 0,C 180,E1 -19143.824,E2 -19143.824} C_VEL
LIN {X 0,Y 249.328,Z 327.373,A -85,B 0,C 180,E1 -19144.959,E2 -19144.959} C_VEL
LIN {X 0,Y 252.142,Z 350.663,A -85,B 0,C 180,E1 -19145.964,E2 -19145.964} C_VEL
LIN {X 0,Y 252.413,Z 356.204,A -85,B 0,C 180,E1 -19146.16,E2 -19146.16} C_VEL
LIN {X 0,Y 251.62,Z 383.873,A -85,B 0,C 180,E1 -19146.982,E2 -19146.982} C_VEL
LIN {X 0,Y 250.822,Z 395.001,A -85,B 0,C 180,E1 -19147.558,E2 -19147.558} C_VEL
LIN {X 0,Y 249.466,Z 406.653,A -85,B 0,C 180,E1 -19148.517,E2 -19148.517} C_VEL
LIN {X 0,Y 248.254,Z 415.346,A -85,B 0,C 180,E1 -19149.493,E2 -19149.493} C_VEL
LIN {X 0,Y 246.866,Z 423.654,A -85,B 0,C 180,E1 -19150.674,E2 -19150.674} C_VEL
LIN {X 0,Y 245.451,Z 431.528,A -85,B 0,C 180,E1 -19152.074,E2 -19152.074} C_VEL
LIN {X 0,Y 244.052,Z 438.899,A -85,B 0,C 180,E1 -19153.695,E2 -19153.695} C_VEL
LIN {X 0,Y 242.596,Z 446.385,A -85,B 0,C 180,E1 -19155.746,E2 -19155.746} C_VEL
LIN {X 0,Y 241.285,Z 453.228,A -85,B 0,C 180,E1 -19158.236,E2 -19158.236} C_VEL
LIN {X 0,Y 240.478,Z 458.444,A -85,B 0,C 180,E1 -19160.751,E2 -19160.751} C_VEL
LIN {X 0,Y 240.036,Z 462.281,A -85,B 0,C 180,E1 -19163.275,E2 -19163.275} C_VEL
LIN {X 0,Y 239.919,Z 464.049,A -85,B 0,C 180,E1 -19164.959,E2 -19164.959} C_VEL
LIN {X 0,Y 239.969,Z 465.321,A -85,B 0,C 180,E1 -19166.643,E2 -19166.643} C_VEL
LIN {X 0,Y 240.036,Z 466.112,A -85,B 0,C 180,E1 -19168.323,E2 -19168.323} C_VEL
LIN {X 0,Y 240.112,Z 466.413,A -85,B 0,C 180,E1 -19170.001,E2 -19170.001} C_VEL
LIN {X 0,Y 240.037,Z 466.104,A -85,B 0,C 180,E1 -19171.679,E2 -19171.679} C_VEL
LIN {X 0,Y 239.97,Z 465.298,A -85,B 0,C 180,E1 -19173.359,E2 -19173.359} C_VEL
LIN {X 0,Y 239.951,Z 463.825,A -85,B 0,C 180,E1 -19175.231,E2 -19175.231} C_VEL
LIN {X 0,Y 240.148,Z 461.055,A -85,B 0,C 180,E1 -19177.568,E2 -19177.568} C_VEL
LIN {X 0,Y 240.478,Z 458.369,A -85,B 0,C 180,E1 -19179.251,E2 -19179.251} C_VEL
LIN {X 0,Y 241.285,Z 453.132,A -85,B 0,C 180,E1 -19181.765,E2 -19181.765} C_VEL
LIN {X 0,Y 242.592,Z 446.243,A -85,B 0,C 180,E1 -19184.256,E2 -19184.256} C_VEL
LIN {X 0,Y 244.036,Z 438.731,A -85,B 0,C 180,E1 -19186.308,E2 -19186.308} C_VEL
LIN {X 0,Y 245.458,Z 431.332,A -85,B 0,C 180,E1 -19187.927,E2 -19187.927} C_VEL
LIN {X 0,Y 246.906,Z 423.414,A -85,B 0,C 180,E1 -19189.324,E2 -19189.324} C_VEL
LIN {X 0,Y 248.465,Z 413.54,A -85,B 0,C 180,E1 -19190.707,E2 -19190.707} C_VEL
LIN {X 0,Y 249.88,Z 402.826,A -85,B 0,C 180,E1 -19191.807,E2 -19191.807} C_VEL
LIN {X 0,Y 250.939,Z 392.673,A -85,B 0,C 180,E1 -19192.541,E2 -19192.541} C_VEL
LIN {X 0,Y 251.584,Z 384.127,A -85,B 0,C 180,E1 -19192.969,E2 -19192.969} C_VEL
LIN {X 0,Y 252.389,Z 354.079,A -85,B 0,C 180,E1 -19193.865,E2 -19193.865} C_VEL
LIN {X 0,Y 249.764,Z 330.902,A -85,B 0,C 180,E1 -19194.842,E2 -19194.842} C_VEL
LIN {X 0,Y 246.464,Z 309.777,A -85,B 0,C 180,E1 -19195.857,E2 -19195.857} C_VEL
LIN {X 0,Y 245.595,Z 304.668,A -85,B 0,C 180,E1 -19196.162,E2 -19196.162} C_VEL
LIN {X 0,Y 245.146,Z 300.55,A -85,B 0,C 180,E1 -19197.766,E2 -19197.766} C_VEL
LIN {X 0,Y 243.477,Z 291.905,A -85,B 0,C 180,E1 -19201.304,E2 -19201.304} C_VEL
LIN {X 0,Y 242.035,Z 285.145,A -85,B 0,C 180,E1 -19204.236,E2 -19204.236} C_VEL
LIN {X 0,Y 241.993,Z 285.154,A -85,B 0,C 180,E1 -19208.359,E2 -19208.359} C_VEL
LIN {X 0,Y 241.901,Z 285.166,A -85,B 0,C 180,E1 -19213.421,E2 -19213.421} C_VEL
LIN {X 0,Y 241.906,Z 285.166,A -85,B 0,C 180,E1 -19218.071,E2 -19218.071} C_VEL
LIN {X 0,Y 241.966,Z 285.16,A -85,B 0,C 180,E1 -19222.414,E2 -19222.414} C_VEL
LIN {X 0,Y 241.98,Z 285.158,A -85,B 0,C 180,E1 -19226.508,E2 -19226.508} C_VEL
LIN {X 0,Y 241.972,Z 285.157,A -85,B 0,C 180,E1 -19230.616,E2 -19230.616} C_VEL
LIN {X 0,Y 241.997,Z 285.156,A -85,B 0,C 180,E1 -19234.198,E2 -19234.198} C_VEL
LIN {X 0,Y 241.987,Z 285.155,A -85,B 0,C 180,E1 -19238.339,E2 -19238.339} C_VEL
LIN {X 0,Y 242.108,Z 285.138,A -85,B 0,C 180,E1 -19243.325,E2 -19243.325} C_VEL
LIN {X 0,Y 242.15,Z 285.13,A -85,B 0,C 180,E1 -19248.278,E2 -19248.278} C_VEL
LIN {X 0,Y 242.36,Z 285.088,A -85,B 0,C 180,E1 -19251.663,E2 -19251.663} C_VEL
LIN {X 0,Y 242.393,Z 285.087,A -85,B 0,C 180,E1 -19253.34,E2 -19253.34} C_VEL
LIN {X 0,Y 242.616,Z 285.074,A -85,B 0,C 180,E1 -19258.34,E2 -19258.34} C_VEL
LIN {X 0,Y 242.618,Z 285.063,A -85,B 0,C 180,E1 -19261.66,E2 -19261.66} C_VEL
LIN {X 0,Y 242.397,Z 285.096,A -85,B 0,C 180,E1 -19266.66,E2 -19266.66} C_VEL
LIN {X 0,Y 242.263,Z 285.118,A -85,B 0,C 180,E1 -19270.024,E2 -19270.024} C_VEL
LIN {X 0,Y 242.109,Z 285.12,A -85,B 0,C 180,E1 -19275.145,E2 -19275.145} C_VEL
LIN {X 0,Y 242.019,Z 285.147,A -85,B 0,C 180,E1 -19278.629,E2 -19278.629} C_VEL
LIN {X 0,Y 241.975,Z 285.154,A -85,B 0,C 180,E1 -19282.184,E2 -19282.184} C_VEL
LIN {X 0,Y 241.989,Z 285.153,A -85,B 0,C 180,E1 -19285.826,E2 -19285.826} C_VEL
LIN {X 0,Y 241.965,Z 285.155,A -85,B 0,C 180,E1 -19289.589,E2 -19289.589} C_VEL
LIN {X 0,Y 241.981,Z 285.146,A -85,B 0,C 180,E1 -19293.493,E2 -19293.493} C_VEL
LIN {X 0,Y 241.967,Z 285.154,A -85,B 0,C 180,E1 -19297.586,E2 -19297.586} C_VEL
LIN {X 0,Y 241.901,Z 285.158,A -85,B 0,C 180,E1 -19301.93,E2 -19301.93} C_VEL
LIN {X 0,Y 241.903,Z 285.166,A -85,B 0,C 180,E1 -19306.579,E2 -19306.579} C_VEL
LIN {X 0,Y 241.996,Z 285.123,A -85,B 0,C 180,E1 -19311.641,E2 -19311.641} C_VEL
LIN {X 0,Y 241.976,Z 285.148,A -85,B 0,C 180,E1 -19314.486,E2 -19314.486} C_VEL
LIN {X 0,Y 241.95,Z 285.159,A -85,B 0,C 180,E1 -19318.475,E2 -19318.475} C_VEL
LIN {X 0,Y 241.958,Z 285.159,A -85,B 0,C 180,E1 -19322.306,E2 -19322.306} C_VEL
LIN {X 0,Y 242.015,Z 285.282,A -85,B 0,C 180,E1 -19323.669,E2 -19323.669} C_VEL
LIN {X 0,Y 243.114,Z 288.158,A -85,B 0,C 180,E1 -19323.892,E2 -19323.892} C_VEL
LIN {X 0,Y 250.168,Z 303.089,A -85,B 0,C 180,E1 -19325.161,E2 -19325.161} C_VEL
LIN {X 0,Y 253.54,Z 311.366,A -85,B 0,C 180,E1 -19325.772,E2 -19325.772} C_VEL
LIN {X 0,Y 252.252,Z 356.136,A -85,B 0,C 180,E1 -19327.041,E2 -19327.041} C_VEL
LIN {X 0,Y 251.893,Z 365.649,A -85,B 0,C 180,E1 -19327.504,E2 -19327.504} C_VEL
LIN {X 0,Y 251.339,Z 374.648,A -85,B 0,C 180,E1 -19328.149,E2 -19328.149} C_VEL
LIN {X 0,Y 250.429,Z 383.906,A -85,B 0,C 180,E1 -19329.033,E2 -19329.033} C_VEL
LIN {X 0,Y 249.061,Z 393.457,A -85,B 0,C 180,E1 -19330.207,E2 -19330.207} C_VEL
LIN {X 0,Y 247.626,Z 403.193,A -85,B 0,C 180,E1 -19331.808,E2 -19331.808} C_VEL
LIN {X 0,Y 246.317,Z 410.885,A -85,B 0,C 180,E1 -19333.421,E2 -19333.421} C_VEL
LIN {X 0,Y 245.065,Z 417.21,A -85,B 0,C 180,E1 -19335.042,E2 -19335.042} C_VEL
LIN {X 0,Y 243.959,Z 422.465,A -85,B 0,C 180,E1 -19336.675,E2 -19336.675} C_VEL
LIN {X 0,Y 243.007,Z 426.85,A -85,B 0,C 180,E1 -19338.319,E2 -19338.319} C_VEL
LIN {X 0,Y 242.259,Z 430.496,A -85,B 0,C 180,E1 -19339.975,E2 -19339.975} C_VEL
LIN {X 0,Y 241.656,Z 433.472,A -85,B 0,C 180,E1 -19341.638,E2 -19341.638} C_VEL
LIN {X 0,Y 241.201,Z 435.775,A -85,B 0,C 180,E1 -19343.306,E2 -19343.306} C_VEL
LIN {X 0,Y 240.732,Z 437.53,A -85,B 0,C 180,E1 -19344.975,E2 -19344.975} C_VEL
LIN {X 0,Y 240.403,Z 438.795,A -85,B 0,C 180,E1 -19346.647,E2 -19346.647} C_VEL
LIN {X 0,Y 240.208,Z 439.592,A -85,B 0,C 180,E1 -19348.323,E2 -19348.323} C_VEL
LIN {X 0,Y 240.147,Z 439.895,A -85,B 0,C 180,E1 -19349.999,E2 -19349.999} C_VEL
LIN {X 0,Y 240.204,Z 439.617,A -85,B 0,C 180,E1 -19351.676,E2 -19351.676} C_VEL
LIN {X 0,Y 240.392,Z 438.871,A -85,B 0,C 180,E1 -19353.351,E2 -19353.351} C_VEL
LIN {X 0,Y 240.727,Z 437.657,A -85,B 0,C 180,E1 -19355.024,E2 -19355.024} C_VEL
LIN {X 0,Y 241.168,Z 435.956,A -85,B 0,C 180,E1 -19356.693,E2 -19356.693} C_VEL
LIN {X 0,Y 241.94,Z 432.235,A -85,B 0,C 180,E1 -19359.192,E2 -19359.192} C_VEL
LIN {X 0,Y 242.998,Z 427.149,A -85,B 0,C 180,E1 -19361.68,E2 -19361.68} C_VEL
LIN {X 0,Y 244.156,Z 421.673,A -85,B 0,C 180,E1 -19363.737,E2 -19363.737} C_VEL
LIN {X 0,Y 245.611,Z 414.781,A -85,B 0,C 180,E1 -19365.773,E2 -19365.773} C_VEL
LIN {X 0,Y 247.12,Z 406.862,A -85,B 0,C 180,E1 -19367.587,E2 -19367.587} C_VEL
LIN {X 0,Y 248.319,Z 399.314,A -85,B 0,C 180,E1 -19368.993,E2 -19368.993} C_VEL
LIN {X 0,Y 249.498,Z 391.392,A -85,B 0,C 180,E1 -19370.185,E2 -19370.185} C_VEL
LIN {X 0,Y 250.608,Z 383.197,A -85,B 0,C 180,E1 -19371.165,E2 -19371.165} C_VEL
LIN {X 0,Y 251.461,Z 374.884,A -85,B 0,C 180,E1 -19371.95,E2 -19371.95} C_VEL
LIN {X 0,Y 251.95,Z 365.892,A -85,B 0,C 180,E1 -19372.607,E2 -19372.607} C_VEL
LIN {X 0,Y 252.355,Z 356.668,A -85,B 0,C 180,E1 -19373.059,E2 -19373.059} C_VEL
LIN {X 0,Y 253.587,Z 311.416,A -85,B 0,C 180,E1 -19374.354,E2 -19374.354} C_VEL
LIN {X 0,Y 246.29,Z 294.601,A -85,B 0,C 180,E1 -19375.671,E2 -19375.671} C_VEL
LIN {X 0,Y 242.125,Z 285.906,A -85,B 0,C 180,E1 -19376.437,E2 -19376.437} C_VEL
LIN {X 0,Y 241.983,Z 285.159,A -85,B 0,C 180,E1 -19376.545,E2 -19376.545} C_VEL
LIN {X 0,Y 241.961,Z 285.158,A -85,B 0,C 180,E1 -19379.588,E2 -19379.588} C_VEL
LIN {X 0,Y 241.977,Z 285.155,A -85,B 0,C 180,E1 -19383.492,E2 -19383.492} C_VEL
LIN {X 0,Y 241.962,Z 285.155,A -85,B 0,C 180,E1 -19387.586,E2 -19387.586} C_VEL
LIN {X 0,Y 241.902,Z 285.156,A -85,B 0,C 180,E1 -19391.929,E2 -19391.929} C_VEL
LIN {X 0,Y 241.896,Z 285.157,A -85,B 0,C 180,E1 -19396.579,E2 -19396.579} C_VEL
LIN {X 0,Y 241.971,Z 285.156,A -85,B 0,C 180,E1 -19401.646,E2 -19401.646} C_VEL
LIN {X 0,Y 241.97,Z 285.153,A -85,B 0,C 180,E1 -19404.486,E2 -19404.486} C_VEL
LIN {X 0,Y 241.945,Z 285.155,A -85,B 0,C 180,E1 -19408.475,E2 -19408.475} C_VEL
LIN {X 0,Y 241.957,Z 285.152,A -85,B 0,C 180,E1 -19412.306,E2 -19412.306} C_VEL
LIN {X 0,Y 242.019,Z 285.148,A -85,B 0,C 180,E1 -19416.012,E2 -19416.012} C_VEL
LIN {X 0,Y 241.98,Z 285.155,A -85,B 0,C 180,E1 -19419.603,E2 -19419.603} C_VEL
LIN {X 0,Y 242.101,Z 285.129,A -85,B 0,C 180,E1 -19423.324,E2 -19423.324} C_VEL
LIN {X 0,Y 242.15,Z 285.128,A -85,B 0,C 180,E1 -19428.278,E2 -19428.278} C_VEL
LIN {X 0,Y 242.363,Z 285.105,A -85,B 0,C 180,E1 -19431.663,E2 -19431.663} C_VEL
LIN {X 0,Y 242.39,Z 285.097,A -85,B 0,C 180,E1 -19433.34,E2 -19433.34} C_VEL
LIN {X 0,Y 242.611,Z 285.065,A -85,B 0,C 180,E1 -19438.34,E2 -19438.34} C_VEL
LIN {X 0,Y 242.611,Z 285.075,A -85,B 0,C 180,E1 -19441.66,E2 -19441.66} C_VEL
LIN {X 0,Y 242.394,Z 285.104,A -85,B 0,C 180,E1 -19446.66,E2 -19446.66} C_VEL
LIN {X 0,Y 242.255,Z 285.119,A -85,B 0,C 180,E1 -19450.024,E2 -19450.024} C_VEL
LIN {X 0,Y 242.099,Z 285.137,A -85,B 0,C 180,E1 -19455.145,E2 -19455.145} C_VEL
LIN {X 0,Y 242.012,Z 285.15,A -85,B 0,C 180,E1 -19458.629,E2 -19458.629} C_VEL
LIN {X 0,Y 241.968,Z 285.158,A -85,B 0,C 180,E1 -19462.184,E2 -19462.184} C_VEL
LIN {X 0,Y 241.975,Z 285.155,A -85,B 0,C 180,E1 -19464.008,E2 -19464.008} C_VEL
LIN {X 0,Y 241.253,Z 285.246,A -85,B 0,C 180,E1 -19465.398,E2 -19465.398} C_VEL
LIN {X 0,Y 238.369,Z 285.608,A -85,B 0,C 180,E1 -19467.664,E2 -19467.664} C_VEL
LIN {X 0,Y 235.962,Z 285.908,A -85,B 0,C 180,E1 -19469.51,E2 -19469.51} C_VEL
LIN {X 0,Y 234.952,Z 286.032,A -85,B 0,C 180,E1 -19470.943,E2 -19470.943} C_VEL
LIN {X 0,Y 234.879,Z 286.036,A -85,B 0,C 180,E1 -19471.428,E2 -19471.428} C_VEL
LIN {X 0,Y 234.917,Z 286.036,A -85,B 0,C 180,E1 -19474.64,E2 -19474.64} C_VEL
LIN {X 0,Y 234.908,Z 286.039,A -85,B 0,C 180,E1 -19478.936,E2 -19478.936} C_VEL
LIN {X 0,Y 234.849,Z 286.047,A -85,B 0,C 180,E1 -19483.495,E2 -19483.495} C_VEL
LIN {X 0,Y 234.849,Z 286.045,A -85,B 0,C 180,E1 -19486.507,E2 -19486.507} C_VEL
LIN {X 0,Y 234.914,Z 286.038,A -85,B 0,C 180,E1 -19491.079,E2 -19491.079} C_VEL
LIN {X 0,Y 234.966,Z 286.139,A -85,B 0,C 180,E1 -19495.18,E2 -19495.18} C_VEL
LIN {X 0,Y 236.672,Z 293.862,A -85,B 0,C 180,E1 -19498.615,E2 -19498.615} C_VEL
LIN {X 0,Y 238.543,Z 303.903,A -85,B 0,C 180,E1 -19502.828,E2 -19502.828} C_VEL
LIN {X 0,Y 238.645,Z 304.519,A -85,B 0,C 180,E1 -19503.024,E2 -19503.024} C_VEL
LIN {X 0,Y 240.147,Z 311.062,A -85,B 0,C 180,E1 -19503.417,E2 -19503.417} C_VEL
LIN {X 0,Y 243.609,Z 333.703,A -85,B 0,C 180,E1 -19504.542,E2 -19504.542} C_VEL
LIN {X 0,Y 245.909,Z 354.256,A -85,B 0,C 180,E1 -19505.439,E2 -19505.439} C_VEL
LIN {X 0,Y 245.097,Z 383.496,A -85,B 0,C 180,E1 -19506.333,E2 -19506.333} C_VEL
LIN {X 0,Y 244.279,Z 394.619,A -85,B 0,C 180,E1 -19506.923,E2 -19506.923} C_VEL
LIN {X 0,Y 242.89,Z 406.268,A -85,B 0,C 180,E1 -19507.905,E2 -19507.905} C_VEL
LIN {X 0,Y 241.584,Z 415.173,A -85,B 0,C 180,E1 -19508.932,E2 -19508.932} C_VEL
LIN {X 0,Y 240.187,Z 423.266,A -85,B 0,C 180,E1 -19510.115,E2 -19510.115} C_VEL
LIN {X 0,Y 238.67,Z 431.137,A -85,B 0,C 180,E1 -19511.547,E2 -19511.547} C_VEL
LIN {X 0,Y 237.236,Z 438.509,A -85,B 0,C 180,E1 -19513.213,E2 -19513.213} C_VEL
LIN {X 0,Y 235.676,Z 445.992,A -85,B 0,C 180,E1 -19515.318,E2 -19515.318} C_VEL
LIN {X 0,Y 234.328,Z 452.837,A -85,B 0,C 180,E1 -19517.882,E2 -19517.882} C_VEL
LIN {X 0,Y 233.449,Z 458.051,A -85,B 0,C 180,E1 -19520.47,E2 -19520.47} C_VEL
LIN {X 0,Y 232.978,Z 461.89,A -85,B 0,C 180,E1 -19523.071,E2 -19523.071} C_VEL
LIN {X 0,Y 232.844,Z 463.75,A -85,B 0,C 180,E1 -19524.903,E2 -19524.903} C_VEL
LIN {X 0,Y 232.864,Z 464.929,A -85,B 0,C 180,E1 -19526.54,E2 -19526.54} C_VEL
LIN {X 0,Y 232.962,Z 465.722,A -85,B 0,C 180,E1 -19528.272,E2 -19528.272} C_VEL
LIN {X 0,Y 233.035,Z 466.022,A -85,B 0,C 180,E1 -19530.001,E2 -19530.001} C_VEL
LIN {X 0,Y 232.963,Z 465.713,A -85,B 0,C 180,E1 -19531.73,E2 -19531.73} C_VEL
LIN {X 0,Y 232.866,Z 464.904,A -85,B 0,C 180,E1 -19533.461,E2 -19533.461} C_VEL
LIN {X 0,Y 232.849,Z 463.617,A -85,B 0,C 180,E1 -19535.196,E2 -19535.196} C_VEL
LIN {X 0,Y 233.084,Z 460.661,A -85,B 0,C 180,E1 -19537.799,E2 -19537.799} C_VEL
LIN {X 0,Y 233.449,Z 457.975,A -85,B 0,C 180,E1 -19539.532,E2 -19539.532} C_VEL
LIN {X 0,Y 234.328,Z 452.738,A -85,B 0,C 180,E1 -19542.12,E2 -19542.12} C_VEL
LIN {X 0,Y 235.67,Z 445.847,A -85,B 0,C 180,E1 -19544.684,E2 -19544.684} C_VEL
LIN {X 0,Y 237.224,Z 438.337,A -85,B 0,C 180,E1 -19546.79,E2 -19546.79} C_VEL
LIN {X 0,Y 238.68,Z 430.935,A -85,B 0,C 180,E1 -19548.454,E2 -19548.454} C_VEL
LIN {X 0,Y 240.212,Z 423.018,A -85,B 0,C 180,E1 -19549.885,E2 -19549.885} C_VEL
LIN {X 0,Y 241.687,Z 413.956,A -85,B 0,C 180,E1 -19551.194,E2 -19551.194} C_VEL
LIN {X 0,Y 243.278,Z 402.58,A -85,B 0,C 180,E1 -19552.416,E2 -19552.416} C_VEL
LIN {X 0,Y 244.413,Z 392.272,A -85,B 0,C 180,E1 -19553.178,E2 -19553.178} C_VEL
LIN {X 0,Y 245.108,Z 382.418,A -85,B 0,C 180,E1 -19553.668,E2 -19553.668} C_VEL
LIN {X 0,Y 245.826,Z 353.828,A -85,B 0,C 180,E1 -19554.538,E2 -19554.538} C_VEL
LIN {X 0,Y 243.21,Z 331.096,A -85,B 0,C 180,E1 -19555.539,E2 -19555.539} C_VEL
LIN {X 0,Y 240.054,Z 310.797,A -85,B 0,C 180,E1 -19556.553,E2 -19556.553} C_VEL
LIN {X 0,Y 238.648,Z 304.532,A -85,B 0,C 180,E1 -19556.925,E2 -19556.925} C_VEL
LIN {X 0,Y 236.978,Z 295.386,A -85,B 0,C 180,E1 -19560.679,E2 -19560.679} C_VEL
LIN {X 0,Y 234.97,Z 286.027,A -85,B 0,C 180,E1 -19564.821,E2 -19564.821} C_VEL
LIN {X 0,Y 234.913,Z 286.037,A -85,B 0,C 180,E1 -19568.936,E2 -19568.936} C_VEL
LIN {X 0,Y 234.854,Z 286.044,A -85,B 0,C 180,E1 -19573.495,E2 -19573.495} C_VEL
LIN {X 0,Y 234.853,Z 286.046,A -85,B 0,C 180,E1 -19576.506,E2 -19576.506} C_VEL
LIN {X 0,Y 234.919,Z 286.037,A -85,B 0,C 180,E1 -19581.079,E2 -19581.079} C_VEL
LIN {X 0,Y 234.923,Z 286.035,A -85,B 0,C 180,E1 -19585.361,E2 -19585.361} C_VEL
LIN {X 0,Y 234.896,Z 286.038,A -85,B 0,C 180,E1 -19589.427,E2 -19589.427} C_VEL
LIN {X 0,Y 234.941,Z 286.033,A -85,B 0,C 180,E1 -19593.822,E2 -19593.822} C_VEL
LIN {X 0,Y 234.936,Z 286.031,A -85,B 0,C 180,E1 -19598.963,E2 -19598.963} C_VEL
LIN {X 0,Y 235.052,Z 286.017,A -85,B 0,C 180,E1 -19603.098,E2 -19603.098} C_VEL
LIN {X 0,Y 235.082,Z 286.012,A -85,B 0,C 180,E1 -19607.921,E2 -19607.921} C_VEL
LIN {X 0,Y 235.298,Z 285.967,A -85,B 0,C 180,E1 -19611.411,E2 -19611.411} C_VEL
LIN {X 0,Y 235.343,Z 285.963,A -85,B 0,C 180,E1 -19613.14,E2 -19613.14} C_VEL
LIN {X 0,Y 235.575,Z 285.951,A -85,B 0,C 180,E1 -19618.291,E2 -19618.291} C_VEL
LIN {X 0,Y 235.577,Z 285.939,A -85,B 0,C 180,E1 -19621.71,E2 -19621.71} C_VEL
LIN {X 0,Y 235.348,Z 285.974,A -85,B 0,C 180,E1 -19626.86,E2 -19626.86} C_VEL
LIN {X 0,Y 235.187,Z 286,A -85,B 0,C 180,E1 -19630.329,E2 -19630.329} C_VEL
LIN {X 0,Y 235.045,Z 286,A -85,B 0,C 180,E1 -19635.611,E2 -19635.611} C_VEL
LIN {X 0,Y 234.96,Z 286.03,A -85,B 0,C 180,E1 -19639.21,E2 -19639.21} C_VEL
LIN {X 0,Y 234.91,Z 286.032,A -85,B 0,C 180,E1 -19642.888,E2 -19642.888} C_VEL
LIN {X 0,Y 234.925,Z 286.033,A -85,B 0,C 180,E1 -19646.663,E2 -19646.663} C_VEL
LIN {X 0,Y 234.897,Z 286.039,A -85,B 0,C 180,E1 -19650.573,E2 -19650.573} C_VEL
LIN {X 0,Y 234.924,Z 286.019,A -85,B 0,C 180,E1 -19654.639,E2 -19654.639} C_VEL
LIN {X 0,Y 234.914,Z 286.036,A -85,B 0,C 180,E1 -19658.935,E2 -19658.935} C_VEL
LIN {X 0,Y 234.861,Z 286.038,A -85,B 0,C 180,E1 -19664.095,E2 -19664.095} C_VEL
LIN {X 0,Y 234.856,Z 286.035,A -85,B 0,C 180,E1 -19668.825,E2 -19668.825} C_VEL
LIN {X 0,Y 234.92,Z 286.004,A -85,B 0,C 180,E1 -19671.078,E2 -19671.078} C_VEL
LIN {X 0,Y 234.925,Z 286.031,A -85,B 0,C 180,E1 -19675.36,E2 -19675.36} C_VEL
LIN {X 0,Y 234.896,Z 286.038,A -85,B 0,C 180,E1 -19679.426,E2 -19679.426} C_VEL
LIN {X 0,Y 234.946,Z 286.033,A -85,B 0,C 180,E1 -19682.797,E2 -19682.797} C_VEL
LIN {X 0,Y 236.014,Z 288.976,A -85,B 0,C 180,E1 -19683.056,E2 -19683.056} C_VEL
LIN {X 0,Y 242.899,Z 303.189,A -85,B 0,C 180,E1 -19684.352,E2 -19684.352} C_VEL
LIN {X 0,Y 247.062,Z 313.028,A -85,B 0,C 180,E1 -19685.134,E2 -19685.134} C_VEL
LIN {X 0,Y 245.733,Z 357.577,A -85,B 0,C 180,E1 -19686.44,E2 -19686.44} C_VEL
LIN {X 0,Y 245.285,Z 367.133,A -85,B 0,C 180,E1 -19686.936,E2 -19686.936} C_VEL
LIN {X 0,Y 244.6,Z 377.641,A -85,B 0,C 180,E1 -19687.754,E2 -19687.754} C_VEL
LIN {X 0,Y 243.349,Z 387.865,A -85,B 0,C 180,E1 -19688.837,E2 -19688.837} C_VEL
LIN {X 0,Y 242.043,Z 396.505,A -85,B 0,C 180,E1 -19690.051,E2 -19690.051} C_VEL
LIN {X 0,Y 240.733,Z 404.602,A -85,B 0,C 180,E1 -19691.488,E2 -19691.488} C_VEL
LIN {X 0,Y 239.529,Z 411.28,A -85,B 0,C 180,E1 -19692.937,E2 -19692.937} C_VEL
LIN {X 0,Y 238.239,Z 417.603,A -85,B 0,C 180,E1 -19694.603,E2 -19694.603} C_VEL
LIN {X 0,Y 237.087,Z 422.857,A -85,B 0,C 180,E1 -19696.281,E2 -19696.281} C_VEL
LIN {X 0,Y 236.072,Z 427.242,A -85,B 0,C 180,E1 -19697.971,E2 -19697.971} C_VEL
LIN {X 0,Y 235.288,Z 430.888,A -85,B 0,C 180,E1 -19699.675,E2 -19699.675} C_VEL
LIN {X 0,Y 234.457,Z 434.733,A -85,B 0,C 180,E1 -19702.021,E2 -19702.021} C_VEL
LIN {X 0,Y 234.161,Z 436.167,A -85,B 0,C 180,E1 -19703.104,E2 -19703.104} C_VEL
LIN {X 0,Y 233.694,Z 437.921,A -85,B 0,C 180,E1 -19704.823,E2 -19704.823} C_VEL
LIN {X 0,Y 233.344,Z 439.186,A -85,B 0,C 180,E1 -19706.546,E2 -19706.546} C_VEL
LIN {X 0,Y 233.136,Z 439.983,A -85,B 0,C 180,E1 -19708.272,E2 -19708.272} C_VEL
LIN {X 0,Y 233.072,Z 440.286,A -85,B 0,C 180,E1 -19709.999,E2 -19709.999} C_VEL
LIN {X 0,Y 233.133,Z 440.008,A -85,B 0,C 180,E1 -19711.727,E2 -19711.727} C_VEL
LIN {X 0,Y 233.334,Z 439.261,A -85,B 0,C 180,E1 -19713.453,E2 -19713.453} C_VEL
LIN {X 0,Y 233.687,Z 438.047,A -85,B 0,C 180,E1 -19715.176,E2 -19715.176} C_VEL
LIN {X 0,Y 234.131,Z 436.347,A -85,B 0,C 180,E1 -19716.895,E2 -19716.895} C_VEL
LIN {X 0,Y 234.914,Z 432.773,A -85,B 0,C 180,E1 -19719.383,E2 -19719.383} C_VEL
LIN {X 0,Y 236.064,Z 427.538,A -85,B 0,C 180,E1 -19722.028,E2 -19722.028} C_VEL
LIN {X 0,Y 237.271,Z 422.062,A -85,B 0,C 180,E1 -19724.143,E2 -19724.143} C_VEL
LIN {X 0,Y 238.801,Z 415.169,A -85,B 0,C 180,E1 -19726.235,E2 -19726.235} C_VEL
LIN {X 0,Y 240.367,Z 407.251,A -85,B 0,C 180,E1 -19728.098,E2 -19728.098} C_VEL
LIN {X 0,Y 241.625,Z 399.702,A -85,B 0,C 180,E1 -19729.541,E2 -19729.541} C_VEL
LIN {X 0,Y 242.862,Z 391.778,A -85,B 0,C 180,E1 -19730.761,E2 -19730.761} C_VEL
LIN {X 0,Y 244.032,Z 383.58,A -85,B 0,C 180,E1 -19731.764,E2 -19731.764} C_VEL
LIN {X 0,Y 244.874,Z 375.436,A -85,B 0,C 180,E1 -19732.557,E2 -19732.557} C_VEL
LIN {X 0,Y 245.452,Z 365.943,A -85,B 0,C 180,E1 -19733.262,E2 -19733.262} C_VEL
LIN {X 0,Y 245.859,Z 357.041,A -85,B 0,C 180,E1 -19733.705,E2 -19733.705} C_VEL
LIN {X 0,Y 247.131,Z 313.124,A -85,B 0,C 180,E1 -19734.991,E2 -19734.991} C_VEL
LIN {X 0,Y 240.106,Z 297.151,A -85,B 0,C 180,E1 -19736.311,E2 -19736.311} C_VEL
LIN {X 0,Y 235.076,Z 286.892,A -85,B 0,C 180,E1 -19737.275,E2 -19737.275} C_VEL
LIN {X 0,Y 234.921,Z 286.037,A -85,B 0,C 180,E1 -19737.328,E2 -19737.328} C_VEL
LIN {X 0,Y 234.893,Z 286.04,A -85,B 0,C 180,E1 -19740.572,E2 -19740.572} C_VEL
LIN {X 0,Y 234.92,Z 286.033,A -85,B 0,C 180,E1 -19744.638,E2 -19744.638} C_VEL
LIN {X 0,Y 234.91,Z 286.035,A -85,B 0,C 180,E1 -19748.934,E2 -19748.934} C_VEL
LIN {X 0,Y 234.849,Z 286.04,A -85,B 0,C 180,E1 -19753.493,E2 -19753.493} C_VEL
LIN {X 0,Y 234.848,Z 286.035,A -85,B 0,C 180,E1 -19756.505,E2 -19756.505} C_VEL
LIN {X 0,Y 234.915,Z 286.032,A -85,B 0,C 180,E1 -19761.078,E2 -19761.078} C_VEL
LIN {X 0,Y 234.918,Z 286.033,A -85,B 0,C 180,E1 -19765.36,E2 -19765.36} C_VEL
LIN {X 0,Y 234.891,Z 286.037,A -85,B 0,C 180,E1 -19769.426,E2 -19769.426} C_VEL
LIN {X 0,Y 234.964,Z 286.029,A -85,B 0,C 180,E1 -19773.806,E2 -19773.806} C_VEL
LIN {X 0,Y 234.961,Z 286.027,A -85,B 0,C 180,E1 -19778.007,E2 -19778.007} C_VEL
LIN {X 0,Y 235.045,Z 286.009,A -85,B 0,C 180,E1 -19783.097,E2 -19783.097} C_VEL
LIN {X 0,Y 235.082,Z 286.008,A -85,B 0,C 180,E1 -19787.92,E2 -19787.92} C_VEL
LIN {X 0,Y 235.3,Z 285.986,A -85,B 0,C 180,E1 -19791.411,E2 -19791.411} C_VEL
LIN {X 0,Y 235.342,Z 285.975,A -85,B 0,C 180,E1 -19793.139,E2 -19793.139} C_VEL
LIN {X 0,Y 235.57,Z 285.941,A -85,B 0,C 180,E1 -19798.29,E2 -19798.29} C_VEL
LIN {X 0,Y 235.57,Z 285.952,A -85,B 0,C 180,E1 -19801.709,E2 -19801.709} C_VEL
LIN {X 0,Y 235.346,Z 285.981,A -85,B 0,C 180,E1 -19806.86,E2 -19806.86} C_VEL
LIN {X 0,Y 235.179,Z 285.999,A -85,B 0,C 180,E1 -19810.329,E2 -19810.329} C_VEL
LIN {X 0,Y 235.052,Z 286.016,A -85,B 0,C 180,E1 -19815.61,E2 -19815.61} C_VEL
LIN {X 0,Y 234.954,Z 286.029,A -85,B 0,C 180,E1 -19819.21,E2 -19819.21} C_VEL
LIN {X 0,Y 234.911,Z 286.035,A -85,B 0,C 180,E1 -19822.888,E2 -19822.888} C_VEL
LIN {X 0,Y 234.917,Z 286.035,A -85,B 0,C 180,E1 -19826.664,E2 -19826.664} C_VEL
LIN {X 0,Y 234.89,Z 286.039,A -85,B 0,C 180,E1 -19830.574,E2 -19830.574} C_VEL
LIN {X 0,Y 234.879,Z 286.036,A -85,B 0,C 180,E1 -19831.428,E2 -19831.428} C_VEL
LIN {X 0,Y 234.23,Z 286.123,A -85,B 0,C 180,E1 -19832.86,E2 -19832.86} C_VEL
LIN {X 0,Y 231.364,Z 286.481,A -85,B 0,C 180,E1 -19835.196,E2 -19835.196} C_VEL
LIN {X 0,Y 228.923,Z 286.785,A -85,B 0,C 180,E1 -19837.101,E2 -19837.101} C_VEL
LIN {X 0,Y 227.887,Z 286.913,A -85,B 0,C 180,E1 -19838.581,E2 -19838.581} C_VEL
LIN {X 0,Y 227.81,Z 286.922,A -85,B 0,C 180,E1 -19839.082,E2 -19839.082} C_VEL
LIN {X 0,Y 227.781,Z 286.926,A -85,B 0,C 180,E1 -19842.749,E2 -19842.749} C_VEL
LIN {X 0,Y 227.782,Z 286.927,A -85,B 0,C 180,E1 -19847.252,E2 -19847.252} C_VEL
LIN {X 0,Y 227.837,Z 286.918,A -85,B 0,C 180,E1 -19851.909,E2 -19851.909} C_VEL
LIN {X 0,Y 227.899,Z 287.028,A -85,B 0,C 180,E1 -19854.532,E2 -19854.532} C_VEL
LIN {X 0,Y 229.649,Z 294.828,A -85,B 0,C 180,E1 -19858.137,E2 -19858.137} C_VEL
LIN {X 0,Y 231.377,Z 303.962,A -85,B 0,C 180,E1 -19862.1,E2 -19862.1} C_VEL
LIN {X 0,Y 233.428,Z 310.228,A -85,B 0,C 180,E1 -19862.574,E2 -19862.574} C_VEL
LIN {X 0,Y 237.077,Z 333.491,A -85,B 0,C 180,E1 -19863.793,E2 -19863.793} C_VEL
LIN {X 0,Y 239.477,Z 355.166,A -85,B 0,C 180,E1 -19864.775,E2 -19864.775} C_VEL
LIN {X 0,Y 238.617,Z 383.12,A -85,B 0,C 180,E1 -19865.649,E2 -19865.649} C_VEL
LIN {X 0,Y 237.834,Z 393.402,A -85,B 0,C 180,E1 -19866.201,E2 -19866.201} C_VEL
LIN {X 0,Y 236.554,Z 404.186,A -85,B 0,C 180,E1 -19867.074,E2 -19867.074} C_VEL
LIN {X 0,Y 235.064,Z 414.263,A -85,B 0,C 180,E1 -19868.239,E2 -19868.239} C_VEL
LIN {X 0,Y 233.533,Z 422.879,A -85,B 0,C 180,E1 -19869.523,E2 -19869.523} C_VEL
LIN {X 0,Y 231.929,Z 430.747,A -85,B 0,C 180,E1 -19870.99,E2 -19870.99} C_VEL
LIN {X 0,Y 230.44,Z 438.119,A -85,B 0,C 180,E1 -19872.702,E2 -19872.702} C_VEL
LIN {X 0,Y 228.786,Z 445.6,A -85,B 0,C 180,E1 -19874.865,E2 -19874.865} C_VEL
LIN {X 0,Y 227.369,Z 452.445,A -85,B 0,C 180,E1 -19877.505,E2 -19877.505} C_VEL
LIN {X 0,Y 226.439,Z 457.66,A -85,B 0,C 180,E1 -19880.172,E2 -19880.172} C_VEL
LIN {X 0,Y 225.915,Z 461.497,A -85,B 0,C 180,E1 -19882.853,E2 -19882.853} C_VEL
LIN {X 0,Y 225.743,Z 463.625,A -85,B 0,C 180,E1 -19885.033,E2 -19885.033} C_VEL
LIN {X 0,Y 225.888,Z 465.331,A -85,B 0,C 180,E1 -19888.218,E2 -19888.218} C_VEL
LIN {X 0,Y 225.961,Z 465.631,A -85,B 0,C 180,E1 -19890.001,E2 -19890.001} C_VEL
LIN {X 0,Y 225.889,Z 465.323,A -85,B 0,C 180,E1 -19891.784,E2 -19891.784} C_VEL
LIN {X 0,Y 225.77,Z 463.513,A -85,B 0,C 180,E1 -19895.046,E2 -19895.046} C_VEL
LIN {X 0,Y 226.042,Z 460.268,A -85,B 0,C 180,E1 -19898.044,E2 -19898.044} C_VEL
LIN {X 0,Y 226.439,Z 457.581,A -85,B 0,C 180,E1 -19899.83,E2 -19899.83} C_VEL
LIN {X 0,Y 227.369,Z 452.343,A -85,B 0,C 180,E1 -19902.497,E2 -19902.497} C_VEL
LIN {X 0,Y 228.78,Z 445.451,A -85,B 0,C 180,E1 -19905.137,E2 -19905.137} C_VEL
LIN {X 0,Y 230.432,Z 437.942,A -85,B 0,C 180,E1 -19907.3,E2 -19907.3} C_VEL
LIN {X 0,Y 231.943,Z 430.539,A -85,B 0,C 180,E1 -19909.011,E2 -19909.011} C_VEL
LIN {X 0,Y 233.553,Z 422.622,A -85,B 0,C 180,E1 -19910.477,E2 -19910.477} C_VEL
LIN {X 0,Y 235.214,Z 412.834,A -85,B 0,C 180,E1 -19911.918,E2 -19911.918} C_VEL
LIN {X 0,Y 236.755,Z 401.689,A -85,B 0,C 180,E1 -19913.116,E2 -19913.116} C_VEL
LIN {X 0,Y 237.892,Z 391.778,A -85,B 0,C 180,E1 -19913.858,E2 -19913.858} C_VEL
LIN {X 0,Y 238.566,Z 383.44,A -85,B 0,C 180,E1 -19914.295,E2 -19914.295} C_VEL
LIN {X 0,Y 239.426,Z 355.704,A -85,B 0,C 180,E1 -19915.166,E2 -19915.166} C_VEL
LIN {X 0,Y 237.064,Z 334.063,A -85,B 0,C 180,E1 -19916.14,E2 -19916.14} C_VEL
LIN {X 0,Y 234.095,Z 314.165,A -85,B 0,C 180,E1 -19917.158,E2 -19917.158} C_VEL
LIN {X 0,Y 232.629,Z 307.394,A -85,B 0,C 180,E1 -19917.57,E2 -19917.57} C_VEL
LIN {X 0,Y 231.332,Z 303.771,A -85,B 0,C 180,E1 -19917.917,E2 -19917.917} C_VEL
LIN {X 0,Y 229.86,Z 295.931,A -85,B 0,C 180,E1 -19921.318,E2 -19921.318} C_VEL
LIN {X 0,Y 227.903,Z 286.909,A -85,B 0,C 180,E1 -19925.467,E2 -19925.467} C_VEL
LIN {X 0,Y 227.828,Z 286.919,A -85,B 0,C 180,E1 -19929.539,E2 -19929.539} C_VEL
LIN {X 0,Y 227.787,Z 286.926,A -85,B 0,C 180,E1 -19932.749,E2 -19932.749} C_VEL
LIN {X 0,Y 227.785,Z 286.926,A -85,B 0,C 180,E1 -19937.252,E2 -19937.252} C_VEL
LIN {X 0,Y 227.839,Z 286.918,A -85,B 0,C 180,E1 -19941.908,E2 -19941.908} C_VEL
LIN {X 0,Y 227.88,Z 286.915,A -85,B 0,C 180,E1 -19946.378,E2 -19946.378} C_VEL
LIN {X 0,Y 227.873,Z 286.914,A -85,B 0,C 180,E1 -19950.431,E2 -19950.431} C_VEL
LIN {X 0,Y 227.873,Z 286.913,A -85,B 0,C 180,E1 -19954.419,E2 -19954.419} C_VEL
LIN {X 0,Y 227.92,Z 286.907,A -85,B 0,C 180,E1 -19958.283,E2 -19958.283} C_VEL
LIN {X 0,Y 228,Z 286.895,A -85,B 0,C 180,E1 -19963.894,E2 -19963.894} C_VEL
LIN {X 0,Y 228.126,Z 286.873,A -85,B 0,C 180,E1 -19969.348,E2 -19969.348} C_VEL
LIN {X 0,Y 228.295,Z 286.839,A -85,B 0,C 180,E1 -19972.927,E2 -19972.927} C_VEL
LIN {X 0,Y 228.533,Z 286.829,A -85,B 0,C 180,E1 -19978.238,E2 -19978.238} C_VEL
LIN {X 0,Y 228.535,Z 286.815,A -85,B 0,C 180,E1 -19981.762,E2 -19981.762} C_VEL
LIN {X 0,Y 228.301,Z 286.853,A -85,B 0,C 180,E1 -19987.073,E2 -19987.073} C_VEL
LIN {X 0,Y 228.128,Z 286.88,A -85,B 0,C 180,E1 -19990.652,E2 -19990.652} C_VEL
LIN {X 0,Y 228.002,Z 286.879,A -85,B 0,C 180,E1 -19996.106,E2 -19996.106} C_VEL
LIN {X 0,Y 227.921,Z 286.904,A -85,B 0,C 180,E1 -20001.717,E2 -20001.717} C_VEL
LIN {X 0,Y 227.904,Z 286.909,A -85,B 0,C 180,E1 -20006.581,E2 -20006.581} C_VEL
LIN {X 0,Y 227.872,Z 286.913,A -85,B 0,C 180,E1 -20010.279,E2 -20010.279} C_VEL
LIN {X 0,Y 227.878,Z 286.901,A -85,B 0,C 180,E1 -20013.721,E2 -20013.721} C_VEL
LIN {X 0,Y 227.839,Z 286.916,A -85,B 0,C 180,E1 -20018.092,E2 -20018.092} C_VEL
LIN {X 0,Y 227.782,Z 286.913,A -85,B 0,C 180,E1 -20022.749,E2 -20022.749} C_VEL
LIN {X 0,Y 227.811,Z 286.921,A -85,B 0,C 180,E1 -20025.199,E2 -20025.199} C_VEL
LIN {X 0,Y 227.803,Z 286.902,A -85,B 0,C 180,E1 -20029.617,E2 -20029.617} C_VEL
LIN {X 0,Y 227.867,Z 286.898,A -85,B 0,C 180,E1 -20034.125,E2 -20034.125} C_VEL
LIN {X 0,Y 227.856,Z 286.915,A -85,B 0,C 180,E1 -20038.375,E2 -20038.375} C_VEL
LIN {X 0,Y 227.865,Z 286.926,A -85,B 0,C 180,E1 -20041.919,E2 -20041.919} C_VEL
LIN {X 0,Y 228.921,Z 289.838,A -85,B 0,C 180,E1 -20042.164,E2 -20042.164} C_VEL
LIN {X 0,Y 235.803,Z 303.536,A -85,B 0,C 180,E1 -20043.518,E2 -20043.518} C_VEL
LIN {X 0,Y 240.626,Z 314.654,A -85,B 0,C 180,E1 -20044.461,E2 -20044.461} C_VEL
LIN {X 0,Y 239.26,Z 357.693,A -85,B 0,C 180,E1 -20045.75,E2 -20045.75} C_VEL
LIN {X 0,Y 238.791,Z 367.46,A -85,B 0,C 180,E1 -20046.266,E2 -20046.266} C_VEL
LIN {X 0,Y 238.069,Z 378.166,A -85,B 0,C 180,E1 -20047.122,E2 -20047.122} C_VEL
LIN {X 0,Y 236.56,Z 389.759,A -85,B 0,C 180,E1 -20048.428,E2 -20048.428} C_VEL
LIN {X 0,Y 235.213,Z 398.123,A -85,B 0,C 180,E1 -20049.674,E2 -20049.674} C_VEL
LIN {X 0,Y 234.027,Z 404.997,A -85,B 0,C 180,E1 -20050.938,E2 -20050.938} C_VEL
LIN {X 0,Y 232.763,Z 411.674,A -85,B 0,C 180,E1 -20052.425,E2 -20052.425} C_VEL
LIN {X 0,Y 231.435,Z 417.995,A -85,B 0,C 180,E1 -20054.138,E2 -20054.138} C_VEL
LIN {X 0,Y 230.202,Z 423.251,A -85,B 0,C 180,E1 -20055.862,E2 -20055.862} C_VEL
LIN {X 0,Y 229.136,Z 427.636,A -85,B 0,C 180,E1 -20057.601,E2 -20057.601} C_VEL
LIN {X 0,Y 228.324,Z 431.28,A -85,B 0,C 180,E1 -20059.356,E2 -20059.356} C_VEL
LIN {X 0,Y 227.39,Z 435.375,A -85,B 0,C 180,E1 -20061.969,E2 -20061.969} C_VEL
LIN {X 0,Y 226.658,Z 438.312,A -85,B 0,C 180,E1 -20064.662,E2 -20064.662} C_VEL
LIN {X 0,Y 226.287,Z 439.576,A -85,B 0,C 180,E1 -20066.438,E2 -20066.438} C_VEL
LIN {X 0,Y 226.066,Z 440.373,A -85,B 0,C 180,E1 -20068.218,E2 -20068.218} C_VEL
LIN {X 0,Y 225.998,Z 440.676,A -85,B 0,C 180,E1 -20069.999,E2 -20069.999} C_VEL
LIN {X 0,Y 226.063,Z 440.398,A -85,B 0,C 180,E1 -20071.781,E2 -20071.781} C_VEL
LIN {X 0,Y 226.277,Z 439.651,A -85,B 0,C 180,E1 -20073.56,E2 -20073.56} C_VEL
LIN {X 0,Y 226.651,Z 438.436,A -85,B 0,C 180,E1 -20075.337,E2 -20075.337} C_VEL
LIN {X 0,Y 227.37,Z 435.595,A -85,B 0,C 180,E1 -20077.995,E2 -20077.995} C_VEL
LIN {X 0,Y 227.948,Z 433.015,A -85,B 0,C 180,E1 -20079.761,E2 -20079.761} C_VEL
LIN {X 0,Y 229.128,Z 427.929,A -85,B 0,C 180,E1 -20082.398,E2 -20082.398} C_VEL
LIN {X 0,Y 230.415,Z 422.451,A -85,B 0,C 180,E1 -20084.573,E2 -20084.573} C_VEL
LIN {X 0,Y 232.01,Z 415.558,A -85,B 0,C 180,E1 -20086.724,E2 -20086.724} C_VEL
LIN {X 0,Y 233.624,Z 407.639,A -85,B 0,C 180,E1 -20088.639,E2 -20088.639} C_VEL
LIN {X 0,Y 234.975,Z 400.088,A -85,B 0,C 180,E1 -20090.117,E2 -20090.117} C_VEL
LIN {X 0,Y 236.268,Z 392.163,A -85,B 0,C 180,E1 -20091.369,E2 -20091.369} C_VEL
LIN {X 0,Y 237.476,Z 383.965,A -85,B 0,C 180,E1 -20092.396,E2 -20092.396} C_VEL
LIN {X 0,Y 238.465,Z 375.023,A -85,B 0,C 180,E1 -20093.274,E2 -20093.274} C_VEL
LIN {X 0,Y 239.013,Z 365.762,A -85,B 0,C 180,E1 -20093.966,E2 -20093.966} C_VEL
LIN {X 0,Y 239.468,Z 355.171,A -85,B 0,C 180,E1 -20094.478,E2 -20094.478} C_VEL
LIN {X 0,Y 240.654,Z 314.759,A -85,B 0,C 180,E1 -20095.671,E2 -20095.671} C_VEL
LIN {X 0,Y 233.714,Z 299.185,A -85,B 0,C 180,E1 -20097.032,E2 -20097.032} C_VEL
LIN {X 0,Y 228.06,Z 287.885,A -85,B 0,C 180,E1 -20098.167,E2 -20098.167} C_VEL
LIN {X 0,Y 227.866,Z 286.914,A -85,B 0,C 180,E1 -20098.253,E2 -20098.253} C_VEL
LIN {X 0,Y 227.852,Z 286.915,A -85,B 0,C 180,E1 -20101.624,E2 -20101.624} C_VEL
LIN {X 0,Y 227.86,Z 286.908,A -85,B 0,C 180,E1 -20105.874,E2 -20105.874} C_VEL
LIN {X 0,Y 227.794,Z 286.915,A -85,B 0,C 180,E1 -20110.382,E2 -20110.382} C_VEL
LIN {X 0,Y 227.806,Z 286.919,A -85,B 0,C 180,E1 -20115.198,E2 -20115.198} C_VEL
LIN {X 0,Y 227.794,Z 286.914,A -85,B 0,C 180,E1 -20119.616,E2 -20119.616} C_VEL
LIN {X 0,Y 227.859,Z 286.911,A -85,B 0,C 180,E1 -20124.124,E2 -20124.124} C_VEL
LIN {X 0,Y 227.85,Z 286.911,A -85,B 0,C 180,E1 -20128.374,E2 -20128.374} C_VEL
LIN {X 0,Y 227.848,Z 286.909,A -85,B 0,C 180,E1 -20132.44,E2 -20132.44} C_VEL
LIN {X 0,Y 227.886,Z 286.908,A -85,B 0,C 180,E1 -20136.364,E2 -20136.364} C_VEL
LIN {X 0,Y 227.886,Z 286.91,A -85,B 0,C 180,E1 -20140.169,E2 -20140.169} C_VEL
LIN {X 0,Y 227.996,Z 286.882,A -85,B 0,C 180,E1 -20143.893,E2 -20143.893} C_VEL
LIN {X 0,Y 228.121,Z 286.881,A -85,B 0,C 180,E1 -20149.347,E2 -20149.347} C_VEL
LIN {X 0,Y 228.294,Z 286.854,A -85,B 0,C 180,E1 -20152.926,E2 -20152.926} C_VEL
LIN {X 0,Y 228.528,Z 286.817,A -85,B 0,C 180,E1 -20158.237,E2 -20158.237} C_VEL
LIN {X 0,Y 228.529,Z 286.829,A -85,B 0,C 180,E1 -20161.762,E2 -20161.762} C_VEL
LIN {X 0,Y 228.299,Z 286.858,A -85,B 0,C 180,E1 -20167.073,E2 -20167.073} C_VEL
LIN {X 0,Y 228.12,Z 286.877,A -85,B 0,C 180,E1 -20170.652,E2 -20170.652} C_VEL
LIN {X 0,Y 228.003,Z 286.894,A -85,B 0,C 180,E1 -20176.106,E2 -20176.106} C_VEL
LIN {X 0,Y 227.914,Z 286.908,A -85,B 0,C 180,E1 -20181.718,E2 -20181.718} C_VEL
LIN {X 0,Y 227.896,Z 286.91,A -85,B 0,C 180,E1 -20186.581,E2 -20186.581} C_VEL
LIN {X 0,Y 227.844,Z 286.918,A -85,B 0,C 180,E1 -20191.438,E2 -20191.438} C_VEL
LIN {X 0,Y 227.858,Z 286.918,A -85,B 0,C 180,E1 -20195.876,E2 -20195.876} C_VEL
LIN {X 0,Y 227.81,Z 286.922,A -85,B 0,C 180,E1 -20199.082,E2 -20199.082} C_VEL
LIN {X 0,Y 227.147,Z 287.008,A -85,B 0,C 180,E1 -20200.558,E2 -20200.558} C_VEL
LIN {X 0,Y 224.258,Z 287.366,A -85,B 0,C 180,E1 -20202.965,E2 -20202.965} C_VEL
LIN {X 0,Y 221.815,Z 287.671,A -85,B 0,C 180,E1 -20204.929,E2 -20204.929} C_VEL
LIN {X 0,Y 220.8,Z 287.796,A -85,B 0,C 180,E1 -20206.456,E2 -20206.456} C_VEL
LIN {X 0,Y 220.736,Z 287.804,A -85,B 0,C 180,E1 -20206.973,E2 -20206.973} C_VEL
LIN {X 0,Y 220.778,Z 287.798,A -85,B 0,C 180,E1 -20210.458,E2 -20210.458} C_VEL
LIN {X 0,Y 220.844,Z 287.809,A -85,B 0,C 180,E1 -20213.793,E2 -20213.793} C_VEL
LIN {X 0,Y 222.619,Z 295.601,A -85,B 0,C 180,E1 -20217.543,E2 -20217.543} C_VEL
LIN {X 0,Y 224.137,Z 303.647,A -85,B 0,C 180,E1 -20221.12,E2 -20221.12} C_VEL
LIN {X 0,Y 227.236,Z 311.93,A -85,B 0,C 180,E1 -20221.833,E2 -20221.833} C_VEL
LIN {X 0,Y 230.781,Z 335.088,A -85,B 0,C 180,E1 -20223.088,E2 -20223.088} C_VEL
LIN {X 0,Y 233.06,Z 356.255,A -85,B 0,C 180,E1 -20224.078,E2 -20224.078} C_VEL
LIN {X 0,Y 232.164,Z 382.744,A -85,B 0,C 180,E1 -20224.926,E2 -20224.926} C_VEL
LIN {X 0,Y 231.285,Z 393.845,A -85,B 0,C 180,E1 -20225.544,E2 -20225.544} C_VEL
LIN {X 0,Y 229.782,Z 405.494,A -85,B 0,C 180,E1 -20226.572,E2 -20226.572} C_VEL
LIN {X 0,Y 228.371,Z 414.483,A -85,B 0,C 180,E1 -20227.663,E2 -20227.663} C_VEL
LIN {X 0,Y 226.891,Z 422.49,A -85,B 0,C 180,E1 -20228.896,E2 -20228.896} C_VEL
LIN {X 0,Y 225.217,Z 430.357,A -85,B 0,C 180,E1 -20230.401,E2 -20230.401} C_VEL
LIN {X 0,Y 223.662,Z 437.729,A -85,B 0,C 180,E1 -20232.161,E2 -20232.161} C_VEL
LIN {X 0,Y 221.925,Z 445.21,A -85,B 0,C 180,E1 -20234.386,E2 -20234.386} C_VEL
LIN {X 0,Y 220.429,Z 452.054,A -85,B 0,C 180,E1 -20237.105,E2 -20237.105} C_VEL
LIN {X 0,Y 219.411,Z 457.267,A -85,B 0,C 180,E1 -20239.854,E2 -20239.854} C_VEL
LIN {X 0,Y 218.849,Z 461.105,A -85,B 0,C 180,E1 -20242.621,E2 -20242.621} C_VEL
LIN {X 0,Y 218.648,Z 463.476,A -85,B 0,C 180,E1 -20245.156,E2 -20245.156} C_VEL
LIN {X 0,Y 218.814,Z 464.94,A -85,B 0,C 180,E1 -20248.16,E2 -20248.16} C_VEL
LIN {X 0,Y 218.888,Z 465.241,A -85,B 0,C 180,E1 -20250.001,E2 -20250.001} C_VEL
LIN {X 0,Y 218.815,Z 464.932,A -85,B 0,C 180,E1 -20251.842,E2 -20251.842} C_VEL
LIN {X 0,Y 218.691,Z 463.329,A -85,B 0,C 180,E1 -20254.975,E2 -20254.975} C_VEL
LIN {X 0,Y 218.853,Z 461.043,A -85,B 0,C 180,E1 -20257.381,E2 -20257.381} C_VEL
LIN {X 0,Y 219.196,Z 458.685,A -85,B 0,C 180,E1 -20259.226,E2 -20259.226} C_VEL
LIN {X 0,Y 220.019,Z 453.881,A -85,B 0,C 180,E1 -20261.984,E2 -20261.984} C_VEL
LIN {X 0,Y 221.085,Z 448.693,A -85,B 0,C 180,E1 -20264.263,E2 -20264.263} C_VEL
LIN {X 0,Y 222.254,Z 443.634,A -85,B 0,C 180,E1 -20266.063,E2 -20266.063} C_VEL
LIN {X 0,Y 223.655,Z 437.547,A -85,B 0,C 180,E1 -20267.842,E2 -20267.842} C_VEL
LIN {X 0,Y 225.234,Z 430.144,A -85,B 0,C 180,E1 -20269.6,E2 -20269.6} C_VEL
LIN {X 0,Y 226.918,Z 422.227,A -85,B 0,C 180,E1 -20271.104,E2 -20271.104} C_VEL
LIN {X 0,Y 228.474,Z 413.291,A -85,B 0,C 180,E1 -20272.465,E2 -20272.465} C_VEL
LIN {X 0,Y 230.166,Z 402.013,A -85,B 0,C 180,E1 -20273.746,E2 -20273.746} C_VEL
LIN {X 0,Y 231.423,Z 391.46,A -85,B 0,C 180,E1 -20274.562,E2 -20274.562} C_VEL
LIN {X 0,Y 232.132,Z 382.517,A -85,B 0,C 180,E1 -20275.037,E2 -20275.037} C_VEL
LIN {X 0,Y 232.925,Z 355.583,A -85,B 0,C 180,E1 -20275.909,E2 -20275.909} C_VEL
LIN {X 0,Y 230.561,Z 333.989,A -85,B 0,C 180,E1 -20276.924,E2 -20276.924} C_VEL
LIN {X 0,Y 227.389,Z 313,A -85,B 0,C 180,E1 -20278.054,E2 -20278.054} C_VEL
LIN {X 0,Y 226.028,Z 308.664,A -85,B 0,C 180,E1 -20278.387,E2 -20278.387} C_VEL
LIN {X 0,Y 224.1,Z 303.426,A -85,B 0,C 180,E1 -20278.856,E2 -20278.856} C_VEL
LIN {X 0,Y 222.587,Z 295.464,A -85,B 0,C 180,E1 -20282.464,E2 -20282.464} C_VEL
LIN {X 0,Y 220.849,Z 287.788,A -85,B 0,C 180,E1 -20286.208,E2 -20286.208} C_VEL
LIN {X 0,Y 220.773,Z 287.798,A -85,B 0,C 180,E1 -20290.182,E2 -20290.182} C_VEL
LIN {X 0,Y 220.754,Z 287.802,A -85,B 0,C 180,E1 -20294.46,E2 -20294.46} C_VEL
LIN {X 0,Y 220.747,Z 287.802,A -85,B 0,C 180,E1 -20298.042,E2 -20298.042} C_VEL
LIN {X 0,Y 220.827,Z 287.794,A -85,B 0,C 180,E1 -20302.794,E2 -20302.794} C_VEL
LIN {X 0,Y 220.813,Z 287.792,A -85,B 0,C 180,E1 -20307.243,E2 -20307.243} C_VEL
LIN {X 0,Y 220.793,Z 287.793,A -85,B 0,C 180,E1 -20311.481,E2 -20311.481} C_VEL
LIN {X 0,Y 220.804,Z 287.792,A -85,B 0,C 180,E1 -20315.558,E2 -20315.558} C_VEL
LIN {X 0,Y 220.846,Z 287.787,A -85,B 0,C 180,E1 -20319.51,E2 -20319.51} C_VEL
LIN {X 0,Y 220.967,Z 287.772,A -85,B 0,C 180,E1 -20323.367,E2 -20323.367} C_VEL
LIN {X 0,Y 221.051,Z 287.756,A -85,B 0,C 180,E1 -20329.003,E2 -20329.003} C_VEL
LIN {X 0,Y 221.232,Z 287.716,A -85,B 0,C 180,E1 -20332.7,E2 -20332.7} C_VEL
LIN {X 0,Y 221.467,Z 287.709,A -85,B 0,C 180,E1 -20338.182,E2 -20338.182} C_VEL
LIN {X 0,Y 221.468,Z 287.694,A -85,B 0,C 180,E1 -20341.819,E2 -20341.819} C_VEL
LIN {X 0,Y 221.238,Z 287.734,A -85,B 0,C 180,E1 -20347.3,E2 -20347.3} C_VEL
LIN {X 0,Y 221.053,Z 287.76,A -85,B 0,C 180,E1 -20350.997,E2 -20350.997} C_VEL
LIN {X 0,Y 220.969,Z 287.756,A -85,B 0,C 180,E1 -20356.634,E2 -20356.634} C_VEL
LIN {X 0,Y 220.848,Z 287.788,A -85,B 0,C 180,E1 -20360.491,E2 -20360.491} C_VEL
LIN {X 0,Y 220.798,Z 287.791,A -85,B 0,C 180,E1 -20364.443,E2 -20364.443} C_VEL
LIN {X 0,Y 220.798,Z 287.79,A -85,B 0,C 180,E1 -20368.519,E2 -20368.519} C_VEL
LIN {X 0,Y 220.813,Z 287.784,A -85,B 0,C 180,E1 -20372.757,E2 -20372.757} C_VEL
LIN {X 0,Y 220.799,Z 287.791,A -85,B 0,C 180,E1 -20377.273,E2 -20377.273} C_VEL
LIN {X 0,Y 220.745,Z 287.791,A -85,B 0,C 180,E1 -20381.959,E2 -20381.959} C_VEL
LIN {X 0,Y 220.755,Z 287.801,A -85,B 0,C 180,E1 -20385.54,E2 -20385.54} C_VEL
LIN {X 0,Y 220.783,Z 287.765,A -85,B 0,C 180,E1 -20390.457,E2 -20390.457} C_VEL
LIN {X 0,Y 220.827,Z 287.757,A -85,B 0,C 180,E1 -20392.793,E2 -20392.793} C_VEL
LIN {X 0,Y 220.813,Z 287.792,A -85,B 0,C 180,E1 -20397.242,E2 -20397.242} C_VEL
LIN {X 0,Y 220.842,Z 287.789,A -85,B 0,C 180,E1 -20400.915,E2 -20400.915} C_VEL
LIN {X 0,Y 221.803,Z 290.62,A -85,B 0,C 180,E1 -20401.2,E2 -20401.2} C_VEL
LIN {X 0,Y 228.571,Z 303.713,A -85,B 0,C 180,E1 -20402.601,E2 -20402.601} C_VEL
LIN {X 0,Y 234.207,Z 316.494,A -85,B 0,C 180,E1 -20403.756,E2 -20403.756} C_VEL
LIN {X 0,Y 232.826,Z 358.271,A -85,B 0,C 180,E1 -20405.042,E2 -20405.042} C_VEL
LIN {X 0,Y 232.289,Z 368.124,A -85,B 0,C 180,E1 -20405.578,E2 -20405.578} C_VEL
LIN {X 0,Y 231.553,Z 378.722,A -85,B 0,C 180,E1 -20406.456,E2 -20406.456} C_VEL
LIN {X 0,Y 229.995,Z 390.154,A -85,B 0,C 180,E1 -20407.78,E2 -20407.78} C_VEL
LIN {X 0,Y 228.595,Z 398.517,A -85,B 0,C 180,E1 -20409.058,E2 -20409.058} C_VEL
LIN {X 0,Y 227.179,Z 406.405,A -85,B 0,C 180,E1 -20410.575,E2 -20410.575} C_VEL
LIN {X 0,Y 226.027,Z 412.068,A -85,B 0,C 180,E1 -20411.883,E2 -20411.883} C_VEL
LIN {X 0,Y 224.645,Z 418.388,A -85,B 0,C 180,E1 -20413.646,E2 -20413.646} C_VEL
LIN {X 0,Y 223.339,Z 423.644,A -85,B 0,C 180,E1 -20415.418,E2 -20415.418} C_VEL
LIN {X 0,Y 222.221,Z 428.029,A -85,B 0,C 180,E1 -20417.209,E2 -20417.209} C_VEL
LIN {X 0,Y 220.999,Z 433.174,A -85,B 0,C 180,E1 -20419.926,E2 -20419.926} C_VEL
LIN {X 0,Y 220.32,Z 436.023,A -85,B 0,C 180,E1 -20421.917,E2 -20421.917} C_VEL
LIN {X 0,Y 219.625,Z 438.703,A -85,B 0,C 180,E1 -20424.49,E2 -20424.49} C_VEL
LIN {X 0,Y 219.233,Z 439.967,A -85,B 0,C 180,E1 -20426.323,E2 -20426.323} C_VEL
LIN {X 0,Y 218.999,Z 440.764,A -85,B 0,C 180,E1 -20428.16,E2 -20428.16} C_VEL
LIN {X 0,Y 218.926,Z 441.067,A -85,B 0,C 180,E1 -20429.999,E2 -20429.999} C_VEL
LIN {X 0,Y 218.995,Z 440.788,A -85,B 0,C 180,E1 -20431.838,E2 -20431.838} C_VEL
LIN {X 0,Y 219.224,Z 440.041,A -85,B 0,C 180,E1 -20433.675,E2 -20433.675} C_VEL
LIN {X 0,Y 219.617,Z 438.826,A -85,B 0,C 180,E1 -20435.508,E2 -20435.508} C_VEL
LIN {X 0,Y 220.295,Z 436.252,A -85,B 0,C 180,E1 -20438.037,E2 -20438.037} C_VEL
LIN {X 0,Y 220.973,Z 433.403,A -85,B 0,C 180,E1 -20440.073,E2 -20440.073} C_VEL
LIN {X 0,Y 222.204,Z 428.319,A -85,B 0,C 180,E1 -20442.79,E2 -20442.79} C_VEL
LIN {X 0,Y 223.58,Z 422.84,A -85,B 0,C 180,E1 -20445.029,E2 -20445.029} C_VEL
LIN {X 0,Y 225.241,Z 415.946,A -85,B 0,C 180,E1 -20447.242,E2 -20447.242} C_VEL
LIN {X 0,Y 226.929,Z 408.027,A -85,B 0,C 180,E1 -20449.21,E2 -20449.21} C_VEL
LIN {X 0,Y 228.355,Z 400.474,A -85,B 0,C 180,E1 -20450.727,E2 -20450.727} C_VEL
LIN {X 0,Y 229.702,Z 392.548,A -85,B 0,C 180,E1 -20452.011,E2 -20452.011} C_VEL
LIN {X 0,Y 230.956,Z 384.349,A -85,B 0,C 180,E1 -20453.065,E2 -20453.065} C_VEL
LIN {X 0,Y 231.909,Z 375.84,A -85,B 0,C 180,E1 -20453.93,E2 -20453.93} C_VEL
LIN {X 0,Y 232.569,Z 366.262,A -85,B 0,C 180,E1 -20454.665,E2 -20454.665} C_VEL
LIN {X 0,Y 233.003,Z 356.86,A -85,B 0,C 180,E1 -20455.143,E2 -20455.143} C_VEL
LIN {X 0,Y 234.241,Z 316.545,A -85,B 0,C 180,E1 -20456.38,E2 -20456.38} C_VEL
LIN {X 0,Y 227.921,Z 302.406,A -85,B 0,C 180,E1 -20457.677,E2 -20457.677} C_VEL
LIN {X 0,Y 220.973,Z 288.629,A -85,B 0,C 180,E1 -20459.143,E2 -20459.143} C_VEL
LIN {X 0,Y 220.808,Z 287.794,A -85,B 0,C 180,E1 -20459.209,E2 -20459.209} C_VEL
LIN {X 0,Y 220.802,Z 287.795,A -85,B 0,C 180,E1 -20464.15,E2 -20464.15} C_VEL
LIN {X 0,Y 220.794,Z 287.791,A -85,B 0,C 180,E1 -20467.272,E2 -20467.272} C_VEL
LIN {X 0,Y 220.743,Z 287.79,A -85,B 0,C 180,E1 -20471.957,E2 -20471.957} C_VEL
LIN {X 0,Y 220.749,Z 287.798,A -85,B 0,C 180,E1 -20475.539,E2 -20475.539} C_VEL
LIN {X 0,Y 220.777,Z 287.793,A -85,B 0,C 180,E1 -20480.456,E2 -20480.456} C_VEL
LIN {X 0,Y 220.822,Z 287.786,A -85,B 0,C 180,E1 -20482.792,E2 -20482.792} C_VEL
LIN {X 0,Y 220.807,Z 287.789,A -85,B 0,C 180,E1 -20487.242,E2 -20487.242} C_VEL
LIN {X 0,Y 220.797,Z 287.79,A -85,B 0,C 180,E1 -20491.481,E2 -20491.481} C_VEL
LIN {X 0,Y 220.841,Z 287.788,A -85,B 0,C 180,E1 -20495.562,E2 -20495.562} C_VEL
LIN {X 0,Y 220.845,Z 287.789,A -85,B 0,C 180,E1 -20499.509,E2 -20499.509} C_VEL
LIN {X 0,Y 220.962,Z 287.759,A -85,B 0,C 180,E1 -20503.366,E2 -20503.366} C_VEL
LIN {X 0,Y 221.046,Z 287.76,A -85,B 0,C 180,E1 -20509.002,E2 -20509.002} C_VEL
LIN {X 0,Y 221.231,Z 287.736,A -85,B 0,C 180,E1 -20512.699,E2 -20512.699} C_VEL
LIN {X 0,Y 221.462,Z 287.696,A -85,B 0,C 180,E1 -20518.181,E2 -20518.181} C_VEL
LIN {X 0,Y 221.462,Z 287.71,A -85,B 0,C 180,E1 -20521.818,E2 -20521.818} C_VEL
LIN {X 0,Y 221.236,Z 287.738,A -85,B 0,C 180,E1 -20527.3,E2 -20527.3} C_VEL
LIN {X 0,Y 221.045,Z 287.759,A -85,B 0,C 180,E1 -20530.997,E2 -20530.997} C_VEL
LIN {X 0,Y 220.965,Z 287.772,A -85,B 0,C 180,E1 -20536.634,E2 -20536.634} C_VEL
LIN {X 0,Y 220.841,Z 287.787,A -85,B 0,C 180,E1 -20540.491,E2 -20540.491} C_VEL
LIN {X 0,Y 220.797,Z 287.791,A -85,B 0,C 180,E1 -20544.443,E2 -20544.443} C_VEL
LIN {X 0,Y 220.79,Z 287.796,A -85,B 0,C 180,E1 -20548.52,E2 -20548.52} C_VEL
LIN {X 0,Y 220.807,Z 287.794,A -85,B 0,C 180,E1 -20552.758,E2 -20552.758} C_VEL
LIN {X 0,Y 220.793,Z 287.798,A -85,B 0,C 180,E1 -20557.274,E2 -20557.274} C_VEL
LIN {X 0,Y 220.743,Z 287.803,A -85,B 0,C 180,E1 -20561.958,E2 -20561.958} C_VEL
LIN {X 0,Y 220.749,Z 287.803,A -85,B 0,C 180,E1 -20565.541,E2 -20565.541} C_VEL
LIN {X 0,Y 220.736,Z 287.804,A -85,B 0,C 180,E1 -20566.973,E2 -20566.973} C_VEL
LIN {X 0,Y 220.072,Z 287.891,A -85,B 0,C 180,E1 -20567.988,E2 -20567.988} C_VEL
LIN {X 0,Y 217.196,Z 288.25,A -85,B 0,C 180,E1 -20569.581,E2 -20569.581} C_VEL
LIN {X 0,Y 214.333,Z 288.602,A -85,B 0,C 180,E1 -20571.215,E2 -20571.215} C_VEL
LIN {X 0,Y 213.731,Z 288.675,A -85,B 0,C 180,E1 -20572.276,E2 -20572.276} C_VEL
LIN {X 0,Y 213.813,Z 288.78,A -85,B 0,C 180,E1 -20573.092,E2 -20573.092} C_VEL
LIN {X 0,Y 215.686,Z 297.021,A -85,B 0,C 180,E1 -20577.215,E2 -20577.215} C_VEL
LIN {X 0,Y 216.844,Z 303.009,A -85,B 0,C 180,E1 -20580.043,E2 -20580.043} C_VEL
LIN {X 0,Y 221.219,Z 314.49,A -85,B 0,C 180,E1 -20581.101,E2 -20581.101} C_VEL
LIN {X 0,Y 224.534,Z 336.885,A -85,B 0,C 180,E1 -20582.353,E2 -20582.353} C_VEL
LIN {X 0,Y 226.666,Z 357.055,A -85,B 0,C 180,E1 -20583.331,E2 -20583.331} C_VEL
LIN {X 0,Y 225.773,Z 382.369,A -85,B 0,C 180,E1 -20584.165,E2 -20584.165} C_VEL
LIN {X 0,Y 224.839,Z 393.462,A -85,B 0,C 180,E1 -20584.794,E2 -20584.794} C_VEL
LIN {X 0,Y 223.275,Z 405.107,A -85,B 0,C 180,E1 -20585.847,E2 -20585.847} C_VEL
LIN {X 0,Y 221.955,Z 413.257,A -85,B 0,C 180,E1 -20586.844,E2 -20586.844} C_VEL
LIN {X 0,Y 220.275,Z 422.101,A -85,B 0,C 180,E1 -20588.23,E2 -20588.23} C_VEL
LIN {X 0,Y 218.535,Z 429.968,A -85,B 0,C 180,E1 -20589.776,E2 -20589.776} C_VEL
LIN {X 0,Y 216.905,Z 437.339,A -85,B 0,C 180,E1 -20591.585,E2 -20591.585} C_VEL
LIN {X 0,Y 215.088,Z 444.819,A -85,B 0,C 180,E1 -20593.876,E2 -20593.876} C_VEL
LIN {X 0,Y 213.475,Z 451.661,A -85,B 0,C 180,E1 -20596.677,E2 -20596.677} C_VEL
LIN {X 0,Y 212.404,Z 456.875,A -85,B 0,C 180,E1 -20599.516,E2 -20599.516} C_VEL
LIN {X 0,Y 211.809,Z 460.714,A -85,B 0,C 180,E1 -20602.374,E2 -20602.374} C_VEL
LIN {X 0,Y 211.558,Z 463.272,A -85,B 0,C 180,E1 -20605.276,E2 -20605.276} C_VEL
LIN {X 0,Y 211.718,Z 464.548,A -85,B 0,C 180,E1 -20608.099,E2 -20608.099} C_VEL
LIN {X 0,Y 211.817,Z 464.85,A -85,B 0,C 180,E1 -20610.001,E2 -20610.001} C_VEL
LIN {X 0,Y 211.718,Z 464.54,A -85,B 0,C 180,E1 -20611.903,E2 -20611.903} C_VEL
LIN {X 0,Y 211.595,Z 463.166,A -85,B 0,C 180,E1 -20614.843,E2 -20614.843} C_VEL
LIN {X 0,Y 211.812,Z 460.65,A -85,B 0,C 180,E1 -20617.628,E2 -20617.628} C_VEL
LIN {X 0,Y 212.405,Z 456.791,A -85,B 0,C 180,E1 -20620.486,E2 -20620.486} C_VEL
LIN {X 0,Y 213.475,Z 451.553,A -85,B 0,C 180,E1 -20623.325,E2 -20623.325} C_VEL
LIN {X 0,Y 215.082,Z 444.662,A -85,B 0,C 180,E1 -20626.127,E2 -20626.127} C_VEL
LIN {X 0,Y 216.898,Z 437.152,A -85,B 0,C 180,E1 -20628.417,E2 -20628.417} C_VEL
LIN {X 0,Y 218.554,Z 429.748,A -85,B 0,C 180,E1 -20630.225,E2 -20630.225} C_VEL
LIN {X 0,Y 220.308,Z 421.831,A -85,B 0,C 180,E1 -20631.769,E2 -20631.769} C_VEL
LIN {X 0,Y 221.863,Z 413.187,A -85,B 0,C 180,E1 -20633.124,E2 -20633.124} C_VEL
LIN {X 0,Y 223.697,Z 401.614,A -85,B 0,C 180,E1 -20634.477,E2 -20634.477} C_VEL
LIN {X 0,Y 224.994,Z 391.058,A -85,B 0,C 180,E1 -20635.313,E2 -20635.313} C_VEL
LIN {X 0,Y 225.687,Z 382.494,A -85,B 0,C 180,E1 -20635.786,E2 -20635.786} C_VEL
LIN {X 0,Y 226.528,Z 356.379,A -85,B 0,C 180,E1 -20636.656,E2 -20636.656} C_VEL
LIN {X 0,Y 224.342,Z 335.868,A -85,B 0,C 180,E1 -20637.653,E2 -20637.653} C_VEL
LIN {X 0,Y 221.262,Z 315.008,A -85,B 0,C 180,E1 -20638.815,E2 -20638.815} C_VEL
LIN {X 0,Y 219.506,Z 309.849,A -85,B 0,C 180,E1 -20639.252,E2 -20639.252} C_VEL
LIN {X 0,Y 216.848,Z 302.943,A -85,B 0,C 180,E1 -20639.927,E2 -20639.927} C_VEL
LIN {X 0,Y 215.233,Z 294.983,A -85,B 0,C 180,E1 -20643.719,E2 -20643.719} C_VEL
LIN {X 0,Y 213.794,Z 288.667,A -85,B 0,C 180,E1 -20646.985,E2 -20646.985} C_VEL
LIN {X 0,Y 213.699,Z 288.68,A -85,B 0,C 180,E1 -20651.129,E2 -20651.129} C_VEL
LIN {X 0,Y 213.702,Z 288.679,A -85,B 0,C 180,E1 -20653.681,E2 -20653.681} C_VEL
LIN {X 0,Y 213.702,Z 288.68,A -85,B 0,C 180,E1 -20656.346,E2 -20656.346} C_VEL
LIN {X 0,Y 213.703,Z 288.68,A -85,B 0,C 180,E1 -20661.329,E2 -20661.329} C_VEL
LIN {X 0,Y 213.755,Z 288.673,A -85,B 0,C 180,E1 -20666.018,E2 -20666.018} C_VEL
LIN {X 0,Y 213.747,Z 288.674,A -85,B 0,C 180,E1 -20670.449,E2 -20670.449} C_VEL
LIN {X 0,Y 213.741,Z 288.672,A -85,B 0,C 180,E1 -20674.694,E2 -20674.694} C_VEL
LIN {X 0,Y 213.776,Z 288.667,A -85,B 0,C 180,E1 -20678.8,E2 -20678.8} C_VEL
LIN {X 0,Y 213.879,Z 288.654,A -85,B 0,C 180,E1 -20682.798,E2 -20682.798} C_VEL
LIN {X 0,Y 213.91,Z 288.651,A -85,B 0,C 180,E1 -20686.704,E2 -20686.704} C_VEL
LIN {X 0,Y 214.126,Z 288.607,A -85,B 0,C 180,E1 -20690.555,E2 -20690.555} C_VEL
LIN {X 0,Y 214.07,Z 288.62,A -85,B 0,C 180,E1 -20694.348,E2 -20694.348} C_VEL
LIN {X 0,Y 214.403,Z 288.589,A -85,B 0,C 180,E1 -20698.122,E2 -20698.122} C_VEL
LIN {X 0,Y 214.514,Z 288.571,A -85,B 0,C 180,E1 -20700,E2 -20700} C_VEL
LIN {X 0,Y 214.405,Z 288.573,A -85,B 0,C 180,E1 -20701.879,E2 -20701.879} C_VEL
LIN {X 0,Y 214.179,Z 288.615,A -85,B 0,C 180,E1 -20707.542,E2 -20707.542} C_VEL
LIN {X 0,Y 213.986,Z 288.638,A -85,B 0,C 180,E1 -20711.365,E2 -20711.365} C_VEL
LIN {X 0,Y 213.87,Z 288.632,A -85,B 0,C 180,E1 -20715.242,E2 -20715.242} C_VEL
LIN {X 0,Y 213.792,Z 288.666,A -85,B 0,C 180,E1 -20719.192,E2 -20719.192} C_VEL
LIN {X 0,Y 213.767,Z 288.665,A -85,B 0,C 180,E1 -20723.236,E2 -20723.236} C_VEL
LIN {X 0,Y 213.788,Z 288.662,A -85,B 0,C 180,E1 -20727.426,E2 -20727.426} C_VEL
LIN {X 0,Y 213.761,Z 288.668,A -85,B 0,C 180,E1 -20731.739,E2 -20731.739} C_VEL
LIN {X 0,Y 213.743,Z 288.661,A -85,B 0,C 180,E1 -20736.289,E2 -20736.289} C_VEL
LIN {X 0,Y 213.697,Z 288.673,A -85,B 0,C 180,E1 -20741.129,E2 -20741.129} C_VEL
LIN {X 0,Y 213.703,Z 288.669,A -85,B 0,C 180,E1 -20743.68,E2 -20743.68} C_VEL
LIN {X 0,Y 213.703,Z 288.681,A -85,B 0,C 180,E1 -20746.345,E2 -20746.345} C_VEL
LIN {X 0,Y 213.705,Z 288.638,A -85,B 0,C 180,E1 -20751.328,E2 -20751.328} C_VEL
LIN {X 0,Y 213.756,Z 288.672,A -85,B 0,C 180,E1 -20756.017,E2 -20756.017} C_VEL
LIN {X 0,Y 213.791,Z 288.668,A -85,B 0,C 180,E1 -20759.883,E2 -20759.883} C_VEL
LIN {X 0,Y 214.946,Z 291.759,A -85,B 0,C 180,E1 -20760.216,E2 -20760.216} C_VEL
LIN {X 0,Y 222.95,Z 307.237,A -85,B 0,C 180,E1 -20761.962,E2 -20761.962} C_VEL
LIN {X 0,Y 227.835,Z 318.274,A -85,B 0,C 180,E1 -20763.01,E2 -20763.01} C_VEL
LIN {X 0,Y 226.443,Z 357.769,A -85,B 0,C 180,E1 -20764.245,E2 -20764.245} C_VEL
LIN {X 0,Y 225.977,Z 367.5,A -85,B 0,C 180,E1 -20764.773,E2 -20764.773} C_VEL
LIN {X 0,Y 225.326,Z 376.262,A -85,B 0,C 180,E1 -20765.473,E2 -20765.473} C_VEL
LIN {X 0,Y 224.278,Z 385.49,A -85,B 0,C 180,E1 -20766.45,E2 -20766.45} C_VEL
LIN {X 0,Y 222.658,Z 395.038,A -85,B 0,C 180,E1 -20767.742,E2 -20767.742} C_VEL
LIN {X 0,Y 220.868,Z 404.772,A -85,B 0,C 180,E1 -20769.511,E2 -20769.511} C_VEL
LIN {X 0,Y 219.318,Z 412.461,A -85,B 0,C 180,E1 -20771.309,E2 -20771.309} C_VEL
LIN {X 0,Y 217.873,Z 418.78,A -85,B 0,C 180,E1 -20773.122,E2 -20773.122} C_VEL
LIN {X 0,Y 216.5,Z 424.036,A -85,B 0,C 180,E1 -20774.947,E2 -20774.947} C_VEL
LIN {X 0,Y 215.326,Z 428.421,A -85,B 0,C 180,E1 -20776.792,E2 -20776.792} C_VEL
LIN {X 0,Y 214.023,Z 433.567,A -85,B 0,C 180,E1 -20779.594,E2 -20779.594} C_VEL
LIN {X 0,Y 213.568,Z 435.429,A -85,B 0,C 180,E1 -20780.833,E2 -20780.833} C_VEL
LIN {X 0,Y 213.08,Z 437.343,A -85,B 0,C 180,E1 -20782.418,E2 -20782.418} C_VEL
LIN {X 0,Y 212.594,Z 439.093,A -85,B 0,C 180,E1 -20784.307,E2 -20784.307} C_VEL
LIN {X 0,Y 212.182,Z 440.358,A -85,B 0,C 180,E1 -20786.201,E2 -20786.201} C_VEL
LIN {X 0,Y 211.933,Z 441.154,A -85,B 0,C 180,E1 -20788.099,E2 -20788.099} C_VEL
LIN {X 0,Y 211.855,Z 441.457,A -85,B 0,C 180,E1 -20789.999,E2 -20789.999} C_VEL
LIN {X 0,Y 211.93,Z 441.178,A -85,B 0,C 180,E1 -20791.899,E2 -20791.899} C_VEL
LIN {X 0,Y 212.173,Z 440.43,A -85,B 0,C 180,E1 -20793.797,E2 -20793.797} C_VEL
LIN {X 0,Y 212.586,Z 439.215,A -85,B 0,C 180,E1 -20795.691,E2 -20795.691} C_VEL
LIN {X 0,Y 213.059,Z 437.516,A -85,B 0,C 180,E1 -20797.581,E2 -20797.581} C_VEL
LIN {X 0,Y 214.01,Z 433.793,A -85,B 0,C 180,E1 -20800.405,E2 -20800.405} C_VEL
LIN {X 0,Y 215.305,Z 428.708,A -85,B 0,C 180,E1 -20803.207,E2 -20803.207} C_VEL
LIN {X 0,Y 216.761,Z 423.228,A -85,B 0,C 180,E1 -20805.514,E2 -20805.514} C_VEL
LIN {X 0,Y 218.497,Z 416.334,A -85,B 0,C 180,E1 -20807.791,E2 -20807.791} C_VEL
LIN {X 0,Y 220.259,Z 408.414,A -85,B 0,C 180,E1 -20809.816,E2 -20809.816} C_VEL
LIN {X 0,Y 221.756,Z 400.86,A -85,B 0,C 180,E1 -20811.373,E2 -20811.373} C_VEL
LIN {X 0,Y 223.166,Z 392.934,A -85,B 0,C 180,E1 -20812.691,E2 -20812.691} C_VEL
LIN {X 0,Y 224.463,Z 384.733,A -85,B 0,C 180,E1 -20813.772,E2 -20813.772} C_VEL
LIN {X 0,Y 225.517,Z 375.628,A -85,B 0,C 180,E1 -20814.713,E2 -20814.713} C_VEL
LIN {X 0,Y 226.168,Z 366.363,A -85,B 0,C 180,E1 -20815.433,E2 -20815.433} C_VEL
LIN {X 0,Y 226.693,Z 355.184,A -85,B 0,C 180,E1 -20815.992,E2 -20815.992} C_VEL
LIN {X 0,Y 227.949,Z 319.47,A -85,B 0,C 180,E1 -20817.078,E2 -20817.078} C_VEL
LIN {X 0,Y 227.391,Z 317.251,A -85,B 0,C 180,E1 -20817.228,E2 -20817.228} C_VEL
LIN {X 0,Y 221.149,Z 303.588,A -85,B 0,C 180,E1 -20818.572,E2 -20818.572} C_VEL
LIN {X 0,Y 214.673,Z 291.304,A -85,B 0,C 180,E1 -20819.998,E2 -20819.998} C_VEL
LIN {X 0,Y 213.794,Z 288.668,A -85,B 0,C 180,E1 -20820.275,E2 -20820.275} C_VEL
LIN {X 0,Y 213.763,Z 288.668,A -85,B 0,C 180,E1 -20824.72,E2 -20824.72} C_VEL
LIN {X 0,Y 213.699,Z 288.678,A -85,B 0,C 180,E1 -20828.67,E2 -20828.67} C_VEL
LIN {X 0,Y 213.698,Z 288.675,A -85,B 0,C 180,E1 -20833.653,E2 -20833.653} C_VEL
LIN {X 0,Y 213.698,Z 288.669,A -85,B 0,C 180,E1 -20836.345,E2 -20836.345} C_VEL
LIN {X 0,Y 213.698,Z 288.675,A -85,B 0,C 180,E1 -20841.328,E2 -20841.328} C_VEL
LIN {X 0,Y 213.75,Z 288.669,A -85,B 0,C 180,E1 -20846.016,E2 -20846.016} C_VEL
LIN {X 0,Y 213.745,Z 288.67,A -85,B 0,C 180,E1 -20850.448,E2 -20850.448} C_VEL
LIN {X 0,Y 213.776,Z 288.668,A -85,B 0,C 180,E1 -20854.698,E2 -20854.698} C_VEL
LIN {X 0,Y 213.773,Z 288.667,A -85,B 0,C 180,E1 -20858.799,E2 -20858.799} C_VEL
LIN {X 0,Y 213.874,Z 288.646,A -85,B 0,C 180,E1 -20862.798,E2 -20862.798} C_VEL
LIN {X 0,Y 213.908,Z 288.634,A -85,B 0,C 180,E1 -20866.704,E2 -20866.704} C_VEL
LIN {X 0,Y 214.124,Z 288.625,A -85,B 0,C 180,E1 -20870.554,E2 -20870.554} C_VEL
LIN {X 0,Y 214.067,Z 288.617,A -85,B 0,C 180,E1 -20874.347,E2 -20874.347} C_VEL
LIN {X 0,Y 214.398,Z 288.575,A -85,B 0,C 180,E1 -20878.121,E2 -20878.121} C_VEL
LIN {X 0,Y 214.507,Z 288.572,A -85,B 0,C 180,E1 -20880,E2 -20880} C_VEL
LIN {X 0,Y 214.399,Z 288.59,A -85,B 0,C 180,E1 -20881.878,E2 -20881.878} C_VEL
LIN {X 0,Y 214.178,Z 288.617,A -85,B 0,C 180,E1 -20887.542,E2 -20887.542} C_VEL
LIN {X 0,Y 213.977,Z 288.639,A -85,B 0,C 180,E1 -20891.365,E2 -20891.365} C_VEL
LIN {X 0,Y 213.866,Z 288.654,A -85,B 0,C 180,E1 -20895.242,E2 -20895.242} C_VEL
LIN {X 0,Y 213.785,Z 288.666,A -85,B 0,C 180,E1 -20899.192,E2 -20899.192} C_VEL
LIN {X 0,Y 213.78,Z 288.668,A -85,B 0,C 180,E1 -20903.235,E2 -20903.235} C_VEL
LIN {X 0,Y 213.781,Z 288.671,A -85,B 0,C 180,E1 -20907.427,E2 -20907.427} C_VEL
LIN {X 0,Y 213.754,Z 288.674,A -85,B 0,C 180,E1 -20911.74,E2 -20911.74} C_VEL
LIN {X 0,Y 213.737,Z 288.676,A -85,B 0,C 180,E1 -20916.289,E2 -20916.289} C_VEL
LIN {X 0,Y 213.693,Z 288.682,A -85,B 0,C 180,E1 -20921.129,E2 -20921.129} C_VEL
LIN {X 0,Y 213.697,Z 288.681,A -85,B 0,C 180,E1 -20923.681,E2 -20923.681} C_VEL
LIN {X 0,Y 213.659,Z 288.681,A -85,B 0,C 180,E1 -20926.952,E2 -20926.952} C_VEL
LIN {X 0,Y 213.701,Z 288.679,A -85,B 0,C 180,E1 -20931.33,E2 -20931.33} C_VEL
LIN {X 0,Y 213.731,Z 288.675,A -85,B 0,C 180,E1 -20932.276,E2 -20932.276} C_VEL
LIN {X 0,Y 213.415,Z 289.341,A -85,B 0,C 180,E1 -20933.139,E2 -20933.139} C_VEL
LIN {X 0,Y 212.097,Z 291.722,A -85,B 0,C 180,E1 -20934.208,E2 -20934.208} C_VEL
LIN {X 0,Y 209.118,Z 296.965,A -85,B 0,C 180,E1 -20936.211,E2 -20936.211} C_VEL
LIN {X 0,Y 208.874,Z 299.018,A -85,B 0,C 180,E1 -20937.152,E2 -20937.152} C_VEL
LIN {X 0,Y 209.558,Z 302.603,A -85,B 0,C 180,E1 -20938.89,E2 -20938.89} C_VEL
LIN {X 0,Y 215.21,Z 316.845,A -85,B 0,C 180,E1 -20940.316,E2 -20940.316} C_VEL
LIN {X 0,Y 218.233,Z 337.698,A -85,B 0,C 180,E1 -20941.526,E2 -20941.526} C_VEL
LIN {X 0,Y 220.264,Z 356.387,A -85,B 0,C 180,E1 -20942.481,E2 -20942.481} C_VEL
LIN {X 0,Y 219.421,Z 381.993,A -85,B 0,C 180,E1 -20943.359,E2 -20943.359} C_VEL
LIN {X 0,Y 218.449,Z 393.08,A -85,B 0,C 180,E1 -20944.003,E2 -20944.003} C_VEL
LIN {X 0,Y 216.818,Z 404.721,A -85,B 0,C 180,E1 -20945.079,E2 -20945.079} C_VEL
LIN {X 0,Y 215.451,Z 412.87,A -85,B 0,C 180,E1 -20946.102,E2 -20946.102} C_VEL
LIN {X 0,Y 213.949,Z 420.479,A -85,B 0,C 180,E1 -20947.297,E2 -20947.297} C_VEL
LIN {X 0,Y 212.139,Z 428.555,A -85,B 0,C 180,E1 -20948.884,E2 -20948.884} C_VEL
LIN {X 0,Y 210.557,Z 435.234,A -85,B 0,C 180,E1 -20950.503,E2 -20950.503} C_VEL
LIN {X 0,Y 208.981,Z 441.582,A -85,B 0,C 180,E1 -20952.383,E2 -20952.383} C_VEL
LIN {X 0,Y 207.593,Z 446.858,A -85,B 0,C 180,E1 -20954.287,E2 -20954.287} C_VEL
LIN {X 0,Y 206.538,Z 451.269,A -85,B 0,C 180,E1 -20956.221,E2 -20956.221} C_VEL
LIN {X 0,Y 205.399,Z 456.483,A -85,B 0,C 180,E1 -20959.154,E2 -20959.154} C_VEL
LIN {X 0,Y 204.739,Z 460.321,A -85,B 0,C 180,E1 -20962.109,E2 -20962.109} C_VEL
LIN {X 0,Y 204.466,Z 463.036,A -85,B 0,C 180,E1 -20965.415,E2 -20965.415} C_VEL
LIN {X 0,Y 204.624,Z 464.157,A -85,B 0,C 180,E1 -20968.033,E2 -20968.033} C_VEL
LIN {X 0,Y 204.747,Z 464.46,A -85,B 0,C 180,E1 -20970.001,E2 -20970.001} C_VEL
LIN {X 0,Y 204.625,Z 464.148,A -85,B 0,C 180,E1 -20971.969,E2 -20971.969} C_VEL
LIN {X 0,Y 204.501,Z 462.949,A -85,B 0,C 180,E1 -20974.706,E2 -20974.706} C_VEL
LIN {X 0,Y 204.741,Z 460.255,A -85,B 0,C 180,E1 -20977.893,E2 -20977.893} C_VEL
LIN {X 0,Y 205.134,Z 457.896,A -85,B 0,C 180,E1 -20979.865,E2 -20979.865} C_VEL
LIN {X 0,Y 206.088,Z 453.091,A -85,B 0,C 180,E1 -20982.808,E2 -20982.808} C_VEL
LIN {X 0,Y 207.314,Z 447.904,A -85,B 0,C 180,E1 -20985.233,E2 -20985.233} C_VEL
LIN {X 0,Y 208.627,Z 442.844,A -85,B 0,C 180,E1 -20987.144,E2 -20987.144} C_VEL
LIN {X 0,Y 210.161,Z 436.756,A -85,B 0,C 180,E1 -20989.03,E2 -20989.03} C_VEL
LIN {X 0,Y 211.906,Z 429.353,A -85,B 0,C 180,E1 -20990.888,E2 -20990.888} C_VEL
LIN {X 0,Y 213.715,Z 421.434,A -85,B 0,C 180,E1 -20992.476,E2 -20992.476} C_VEL
LIN {X 0,Y 215.411,Z 412.509,A -85,B 0,C 180,E1 -20993.907,E2 -20993.907} C_VEL
LIN {X 0,Y 217.258,Z 401.215,A -85,B 0,C 180,E1 -20995.253,E2 -20995.253} C_VEL
LIN {X 0,Y 218.613,Z 390.657,A -85,B 0,C 180,E1 -20996.107,E2 -20996.107} C_VEL
LIN {X 0,Y 219.315,Z 382.086,A -85,B 0,C 180,E1 -20996.593,E2 -20996.593} C_VEL
LIN {X 0,Y 220.18,Z 357.174,A -85,B 0,C 180,E1 -20997.445,E2 -20997.445} C_VEL
LIN {X 0,Y 218.048,Z 336.873,A -85,B 0,C 180,E1 -20998.471,E2 -20998.471} C_VEL
LIN {X 0,Y 215.199,Z 317.105,A -85,B 0,C 180,E1 -20999.613,E2 -20999.613} C_VEL
LIN {X 0,Y 212.267,Z 309.281,A -85,B 0,C 180,E1 -21000.356,E2 -21000.356} C_VEL
LIN {X 0,Y 209.576,Z 302.458,A -85,B 0,C 180,E1 -21001.089,E2 -21001.089} C_VEL
LIN {X 0,Y 207.89,Z 294.498,A -85,B 0,C 180,E1 -21005.08,E2 -21005.08} C_VEL
LIN {X 0,Y 206.686,Z 289.552,A -85,B 0,C 180,E1 -21007.74,E2 -21007.74} C_VEL
LIN {X 0,Y 206.632,Z 289.56,A -85,B 0,C 180,E1 -21011.56,E2 -21011.56} C_VEL
LIN {X 0,Y 206.631,Z 289.56,A -85,B 0,C 180,E1 -21015.584,E2 -21015.584} C_VEL
LIN {X 0,Y 206.647,Z 289.559,A -85,B 0,C 180,E1 -21019.746,E2 -21019.746} C_VEL
LIN {X 0,Y 206.701,Z 289.553,A -85,B 0,C 180,E1 -21024.689,E2 -21024.689} C_VEL
LIN {X 0,Y 206.696,Z 289.551,A -85,B 0,C 180,E1 -21029.335,E2 -21029.335} C_VEL
LIN {X 0,Y 206.681,Z 289.554,A -85,B 0,C 180,E1 -21033.765,E2 -21033.765} C_VEL
LIN {X 0,Y 206.715,Z 289.551,A -85,B 0,C 180,E1 -21038.039,E2 -21038.039} C_VEL
LIN {X 0,Y 206.805,Z 289.538,A -85,B 0,C 180,E1 -21042.191,E2 -21042.191} C_VEL
LIN {X 0,Y 206.851,Z 289.531,A -85,B 0,C 180,E1 -21046.242,E2 -21046.242} C_VEL
LIN {X 0,Y 207.074,Z 289.486,A -85,B 0,C 180,E1 -21050.23,E2 -21050.23} C_VEL
LIN {X 0,Y 207.033,Z 289.492,A -85,B 0,C 180,E1 -21054.155,E2 -21054.155} C_VEL
LIN {X 0,Y 207.343,Z 289.469,A -85,B 0,C 180,E1 -21058.058,E2 -21058.058} C_VEL
LIN {X 0,Y 207.482,Z 289.446,A -85,B 0,C 180,E1 -21060,E2 -21060} C_VEL
LIN {X 0,Y 207.344,Z 289.452,A -85,B 0,C 180,E1 -21061.943,E2 -21061.943} C_VEL
LIN {X 0,Y 207.124,Z 289.495,A -85,B 0,C 180,E1 -21067.801,E2 -21067.801} C_VEL
LIN {X 0,Y 206.906,Z 289.518,A -85,B 0,C 180,E1 -21071.76,E2 -21071.76} C_VEL
LIN {X 0,Y 206.803,Z 289.513,A -85,B 0,C 180,E1 -21075.776,E2 -21075.776} C_VEL
LIN {X 0,Y 206.713,Z 289.547,A -85,B 0,C 180,E1 -21079.876,E2 -21079.876} C_VEL
LIN {X 0,Y 206.694,Z 289.546,A -85,B 0,C 180,E1 -21084.081,E2 -21084.081} C_VEL
LIN {X 0,Y 206.689,Z 289.546,A -85,B 0,C 180,E1 -21088.427,E2 -21088.427} C_VEL
LIN {X 0,Y 206.696,Z 289.541,A -85,B 0,C 180,E1 -21092.958,E2 -21092.958} C_VEL
LIN {X 0,Y 206.702,Z 289.531,A -85,B 0,C 180,E1 -21095.311,E2 -21095.311} C_VEL
LIN {X 0,Y 206.647,Z 289.555,A -85,B 0,C 180,E1 -21100.255,E2 -21100.255} C_VEL
LIN {X 0,Y 206.631,Z 289.555,A -85,B 0,C 180,E1 -21104.417,E2 -21104.417} C_VEL
LIN {X 0,Y 206.633,Z 289.55,A -85,B 0,C 180,E1 -21108.44,E2 -21108.44} C_VEL
LIN {X 0,Y 206.669,Z 289.513,A -85,B 0,C 180,E1 -21112.257,E2 -21112.257} C_VEL
LIN {X 0,Y 206.696,Z 289.55,A -85,B 0,C 180,E1 -21117.041,E2 -21117.041} C_VEL
LIN {X 0,Y 206.754,Z 289.579,A -85,B 0,C 180,E1 -21118.798,E2 -21118.798} C_VEL
LIN {X 0,Y 207.716,Z 292.35,A -85,B 0,C 180,E1 -21119.071,E2 -21119.071} C_VEL
LIN {X 0,Y 210.681,Z 297.656,A -85,B 0,C 180,E1 -21119.767,E2 -21119.767} C_VEL
LIN {X 0,Y 218.557,Z 313.238,A -85,B 0,C 180,E1 -21121.557,E2 -21121.557} C_VEL
LIN {X 0,Y 221.523,Z 320.546,A -85,B 0,C 180,E1 -21122.243,E2 -21122.243} C_VEL
LIN {X 0,Y 220.093,Z 358.177,A -85,B 0,C 180,E1 -21123.445,E2 -21123.445} C_VEL
LIN {X 0,Y 219.619,Z 367.587,A -85,B 0,C 180,E1 -21123.964,E2 -21123.964} C_VEL
LIN {X 0,Y 219.065,Z 375.004,A -85,B 0,C 180,E1 -21124.549,E2 -21124.549} C_VEL
LIN {X 0,Y 218.069,Z 384.022,A -85,B 0,C 180,E1 -21125.484,E2 -21125.484} C_VEL
LIN {X 0,Y 216.679,Z 392.442,A -85,B 0,C 180,E1 -21126.588,E2 -21126.588} C_VEL
LIN {X 0,Y 215.444,Z 399.306,A -85,B 0,C 180,E1 -21127.714,E2 -21127.714} C_VEL
LIN {X 0,Y 213.877,Z 407.193,A -85,B 0,C 180,E1 -21129.313,E2 -21129.313} C_VEL
LIN {X 0,Y 212.63,Z 412.854,A -85,B 0,C 180,E1 -21130.698,E2 -21130.698} C_VEL
LIN {X 0,Y 211.119,Z 419.173,A -85,B 0,C 180,E1 -21132.565,E2 -21132.565} C_VEL
LIN {X 0,Y 209.658,Z 424.43,A -85,B 0,C 180,E1 -21134.444,E2 -21134.444} C_VEL
LIN {X 0,Y 208.452,Z 428.813,A -85,B 0,C 180,E1 -21136.348,E2 -21136.348} C_VEL
LIN {X 0,Y 207.061,Z 433.959,A -85,B 0,C 180,E1 -21139.24,E2 -21139.24} C_VEL
LIN {X 0,Y 206.474,Z 436.139,A -85,B 0,C 180,E1 -21140.791,E2 -21140.791} C_VEL
LIN {X 0,Y 206.063,Z 437.735,A -85,B 0,C 180,E1 -21142.158,E2 -21142.158} C_VEL
LIN {X 0,Y 205.544,Z 439.485,A -85,B 0,C 180,E1 -21144.111,E2 -21144.111} C_VEL
LIN {X 0,Y 205.133,Z 440.748,A -85,B 0,C 180,E1 -21146.07,E2 -21146.07} C_VEL
LIN {X 0,Y 204.87,Z 441.545,A -85,B 0,C 180,E1 -21148.033,E2 -21148.033} C_VEL
LIN {X 0,Y 204.787,Z 441.848,A -85,B 0,C 180,E1 -21149.999,E2 -21149.999} C_VEL
LIN {X 0,Y 204.866,Z 441.568,A -85,B 0,C 180,E1 -21151.965,E2 -21151.965} C_VEL
LIN {X 0,Y 205.125,Z 440.82,A -85,B 0,C 180,E1 -21153.928,E2 -21153.928} C_VEL
LIN {X 0,Y 205.535,Z 439.606,A -85,B 0,C 180,E1 -21155.887,E2 -21155.887} C_VEL
LIN {X 0,Y 206.044,Z 437.906,A -85,B 0,C 180,E1 -21157.841,E2 -21157.841} C_VEL
LIN {X 0,Y 207.035,Z 434.183,A -85,B 0,C 180,E1 -21160.759,E2 -21160.759} C_VEL
LIN {X 0,Y 208.428,Z 429.097,A -85,B 0,C 180,E1 -21163.651,E2 -21163.651} C_VEL
LIN {X 0,Y 209.958,Z 423.616,A -85,B 0,C 180,E1 -21166.03,E2 -21166.03} C_VEL
LIN {X 0,Y 211.777,Z 416.721,A -85,B 0,C 180,E1 -21168.376,E2 -21168.376} C_VEL
LIN {X 0,Y 213.614,Z 408.802,A -85,B 0,C 180,E1 -21170.46,E2 -21170.46} C_VEL
LIN {X 0,Y 215.188,Z 401.246,A -85,B 0,C 180,E1 -21172.059,E2 -21172.059} C_VEL
LIN {X 0,Y 216.667,Z 393.319,A -85,B 0,C 180,E1 -21173.412,E2 -21173.412} C_VEL
LIN {X 0,Y 218.002,Z 385.118,A -85,B 0,C 180,E1 -21174.522,E2 -21174.522} C_VEL
LIN {X 0,Y 219.082,Z 376.362,A -85,B 0,C 180,E1 -21175.453,E2 -21175.453} C_VEL
LIN {X 0,Y 219.78,Z 366.859,A -85,B 0,C 180,E1 -21176.218,E2 -21176.218} C_VEL
LIN {X 0,Y 220.354,Z 355.98,A -85,B 0,C 180,E1 -21176.777,E2 -21176.777} C_VEL
LIN {X 0,Y 221.572,Z 320.31,A -85,B 0,C 180,E1 -21177.907,E2 -21177.907} C_VEL
LIN {X 0,Y 215.082,Z 306.17,A -85,B 0,C 180,E1 -21179.373,E2 -21179.373} C_VEL
LIN {X 0,Y 208.076,Z 292.854,A -85,B 0,C 180,E1 -21181.007,E2 -21181.007} C_VEL
LIN {X 0,Y 206.941,Z 290.604,A -85,B 0,C 180,E1 -21181.288,E2 -21181.288} C_VEL
LIN {X 0,Y 206.723,Z 289.548,A -85,B 0,C 180,E1 -21181.418,E2 -21181.418} C_VEL
LIN {X 0,Y 206.698,Z 289.544,A -85,B 0,C 180,E1 -21185.31,E2 -21185.31} C_VEL
LIN {X 0,Y 206.643,Z 289.549,A -85,B 0,C 180,E1 -21190.254,E2 -21190.254} C_VEL
LIN {X 0,Y 206.626,Z 289.558,A -85,B 0,C 180,E1 -21194.416,E2 -21194.416} C_VEL
LIN {X 0,Y 206.627,Z 289.543,A -85,B 0,C 180,E1 -21198.44,E2 -21198.44} C_VEL
LIN {X 0,Y 206.661,Z 289.551,A -85,B 0,C 180,E1 -21202.256,E2 -21202.256} C_VEL
LIN {X 0,Y 206.696,Z 289.546,A -85,B 0,C 180,E1 -21204.688,E2 -21204.688} C_VEL
LIN {X 0,Y 206.692,Z 289.549,A -85,B 0,C 180,E1 -21209.334,E2 -21209.334} C_VEL
LIN {X 0,Y 206.7,Z 289.55,A -85,B 0,C 180,E1 -21213.767,E2 -21213.767} C_VEL
LIN {X 0,Y 206.712,Z 289.545,A -85,B 0,C 180,E1 -21218.038,E2 -21218.038} C_VEL
LIN {X 0,Y 206.799,Z 289.532,A -85,B 0,C 180,E1 -21222.19,E2 -21222.19} C_VEL
LIN {X 0,Y 206.848,Z 289.511,A -85,B 0,C 180,E1 -21226.241,E2 -21226.241} C_VEL
LIN {X 0,Y 207.069,Z 289.503,A -85,B 0,C 180,E1 -21230.229,E2 -21230.229} C_VEL
LIN {X 0,Y 207.03,Z 289.494,A -85,B 0,C 180,E1 -21234.155,E2 -21234.155} C_VEL
LIN {X 0,Y 207.338,Z 289.453,A -85,B 0,C 180,E1 -21238.057,E2 -21238.057} C_VEL
LIN {X 0,Y 207.475,Z 289.448,A -85,B 0,C 180,E1 -21240,E2 -21240} C_VEL
LIN {X 0,Y 207.338,Z 289.47,A -85,B 0,C 180,E1 -21241.942,E2 -21241.942} C_VEL
LIN {X 0,Y 207.122,Z 289.497,A -85,B 0,C 180,E1 -21247.8,E2 -21247.8} C_VEL
LIN {X 0,Y 206.898,Z 289.521,A -85,B 0,C 180,E1 -21251.76,E2 -21251.76} C_VEL
LIN {X 0,Y 206.799,Z 289.534,A -85,B 0,C 180,E1 -21255.776,E2 -21255.776} C_VEL
LIN {X 0,Y 206.706,Z 289.547,A -85,B 0,C 180,E1 -21259.877,E2 -21259.877} C_VEL
LIN {X 0,Y 206.696,Z 289.548,A -85,B 0,C 180,E1 -21264.08,E2 -21264.08} C_VEL
LIN {X 0,Y 206.681,Z 289.554,A -85,B 0,C 180,E1 -21268.428,E2 -21268.428} C_VEL
LIN {X 0,Y 206.689,Z 289.554,A -85,B 0,C 180,E1 -21272.959,E2 -21272.959} C_VEL
LIN {X 0,Y 206.696,Z 289.554,A -85,B 0,C 180,E1 -21275.312,E2 -21275.312} C_VEL
LIN {X 0,Y 206.642,Z 289.56,A -85,B 0,C 180,E1 -21280.255,E2 -21280.255} C_VEL
LIN {X 0,Y 206.625,Z 289.562,A -85,B 0,C 180,E1 -21284.418,E2 -21284.418} C_VEL
LIN {X 0,Y 206.627,Z 289.561,A -85,B 0,C 180,E1 -21288.442,E2 -21288.442} C_VEL
LIN {X 0,Y 206.693,Z 289.637,A -85,B 0,C 180,E1 -21292.264,E2 -21292.264} C_VEL
LIN {X 0,Y 208.751,Z 298.382,A -85,B 0,C 180,E1 -21296.835,E2 -21296.835} C_VEL
LIN {X 0,Y 208.874,Z 299.018,A -85,B 0,C 180,E1 -21297.152,E2 -21297.152} C_VEL
LIN {X 0,Y 209.232,Z 301.419,A -85,B 0,C 180,E1 -21297.966,E2 -21297.966} C_VEL
LIN {X 0,Y 209.604,Z 305.45,A -85,B 0,C 180,E1 -21298.7,E2 -21298.7} C_VEL
LIN {X 0,Y 209.854,Z 310.085,A -85,B 0,C 180,E1 -21299.18,E2 -21299.18} C_VEL
LIN {X 0,Y 210.333,Z 324.681,A -85,B 0,C 180,E1 -21299.865,E2 -21299.865} C_VEL
LIN {X 0,Y 210.715,Z 328.85,A -85,B 0,C 180,E1 -21300.089,E2 -21300.089} C_VEL
LIN {X 0,Y 213.56,Z 353.161,A -85,B 0,C 180,E1 -21301.434,E2 -21301.434} C_VEL
LIN {X 0,Y 213.978,Z 358.896,A -85,B 0,C 180,E1 -21301.707,E2 -21301.707} C_VEL
LIN {X 0,Y 213.065,Z 381.615,A -85,B 0,C 180,E1 -21302.498,E2 -21302.498} C_VEL
LIN {X 0,Y 212.092,Z 392.698,A -85,B 0,C 180,E1 -21303.162,E2 -21303.162} C_VEL
LIN {X 0,Y 210.384,Z 404.334,A -85,B 0,C 180,E1 -21304.262,E2 -21304.262} C_VEL
LIN {X 0,Y 208.976,Z 412.482,A -85,B 0,C 180,E1 -21305.313,E2 -21305.313} C_VEL
LIN {X 0,Y 207.399,Z 420.09,A -85,B 0,C 180,E1 -21306.538,E2 -21306.538} C_VEL
LIN {X 0,Y 205.539,Z 428.167,A -85,B 0,C 180,E1 -21308.172,E2 -21308.172} C_VEL
LIN {X 0,Y 203.855,Z 434.843,A -85,B 0,C 180,E1 -21309.834,E2 -21309.834} C_VEL
LIN {X 0,Y 202.213,Z 441.191,A -85,B 0,C 180,E1 -21311.773,E2 -21311.773} C_VEL
LIN {X 0,Y 200.752,Z 446.467,A -85,B 0,C 180,E1 -21313.737,E2 -21313.737} C_VEL
LIN {X 0,Y 199.618,Z 450.876,A -85,B 0,C 180,E1 -21315.734,E2 -21315.734} C_VEL
LIN {X 0,Y 198.389,Z 456.089,A -85,B 0,C 180,E1 -21318.766,E2 -21318.766} C_VEL
LIN {X 0,Y 197.692,Z 459.929,A -85,B 0,C 180,E1 -21321.826,E2 -21321.826} C_VEL
LIN {X 0,Y 197.375,Z 462.794,A -85,B 0,C 180,E1 -21325.561,E2 -21325.561} C_VEL
LIN {X 0,Y 197.531,Z 463.765,A -85,B 0,C 180,E1 -21327.962,E2 -21327.962} C_VEL
LIN {X 0,Y 197.677,Z 464.07,A -85,B 0,C 180,E1 -21330.001,E2 -21330.001} C_VEL
LIN {X 0,Y 197.533,Z 463.756,A -85,B 0,C 180,E1 -21332.04,E2 -21332.04} C_VEL
LIN {X 0,Y 197.404,Z 462.717,A -85,B 0,C 180,E1 -21334.544,E2 -21334.544} C_VEL
LIN {X 0,Y 197.693,Z 459.861,A -85,B 0,C 180,E1 -21338.176,E2 -21338.176} C_VEL
LIN {X 0,Y 198.132,Z 457.503,A -85,B 0,C 180,E1 -21340.217,E2 -21340.217} C_VEL
LIN {X 0,Y 199.15,Z 452.696,A -85,B 0,C 180,E1 -21343.262,E2 -21343.262} C_VEL
LIN {X 0,Y 200.457,Z 447.509,A -85,B 0,C 180,E1 -21345.767,E2 -21345.767} C_VEL
LIN {X 0,Y 201.816,Z 442.448,A -85,B 0,C 180,E1 -21347.742,E2 -21347.742} C_VEL
LIN {X 0,Y 203.431,Z 436.36,A -85,B 0,C 180,E1 -21349.685,E2 -21349.685} C_VEL
LIN {X 0,Y 205.028,Z 429.983,A -85,B 0,C 180,E1 -21351.36,E2 -21351.36} C_VEL
LIN {X 0,Y 206.914,Z 422.274,A -85,B 0,C 180,E1 -21352.993,E2 -21352.993} C_VEL
LIN {X 0,Y 208.397,Z 414.73,A -85,B 0,C 180,E1 -21354.303,E2 -21354.303} C_VEL
LIN {X 0,Y 210.086,Z 405.602,A -85,B 0,C 180,E1 -21355.537,E2 -21355.537} C_VEL
LIN {X 0,Y 211.54,Z 395.971,A -85,B 0,C 180,E1 -21356.516,E2 -21356.516} C_VEL
LIN {X 0,Y 212.884,Z 383.7,A -85,B 0,C 180,E1 -21357.359,E2 -21357.359} C_VEL
LIN {X 0,Y 213.625,Z 366.705,A -85,B 0,C 180,E1 -21357.991,E2 -21357.991} C_VEL
LIN {X 0,Y 213.793,Z 356.753,A -85,B 0,C 180,E1 -21358.337,E2 -21358.337} C_VEL
LIN {X 0,Y 211.514,Z 335.659,A -85,B 0,C 180,E1 -21359.465,E2 -21359.465} C_VEL
LIN {X 0,Y 209.179,Z 319.226,A -85,B 0,C 180,E1 -21360.457,E2 -21360.457} C_VEL
LIN {X 0,Y 203.744,Z 305.687,A -85,B 0,C 180,E1 -21361.892,E2 -21361.892} C_VEL
LIN {X 0,Y 202.278,Z 302.076,A -85,B 0,C 180,E1 -21362.299,E2 -21362.299} C_VEL
LIN {X 0,Y 200.528,Z 294.002,A -85,B 0,C 180,E1 -21366.571,E2 -21366.571} C_VEL
LIN {X 0,Y 199.635,Z 290.431,A -85,B 0,C 180,E1 -21368.674,E2 -21368.674} C_VEL
LIN {X 0,Y 199.567,Z 290.44,A -85,B 0,C 180,E1 -21372.308,E2 -21372.308} C_VEL
LIN {X 0,Y 199.577,Z 290.44,A -85,B 0,C 180,E1 -21375.228,E2 -21375.228} C_VEL
LIN {X 0,Y 199.57,Z 290.44,A -85,B 0,C 180,E1 -21378.003,E2 -21378.003} C_VEL
LIN {X 0,Y 199.597,Z 290.438,A -85,B 0,C 180,E1 -21380.774,E2 -21380.774} C_VEL
LIN {X 0,Y 199.612,Z 290.434,A -85,B 0,C 180,E1 -21385.714,E2 -21385.714} C_VEL
LIN {X 0,Y 199.687,Z 290.423,A -85,B 0,C 180,E1 -21388.135,E2 -21388.135} C_VEL
LIN {X 0,Y 199.627,Z 290.432,A -85,B 0,C 180,E1 -21392.763,E2 -21392.763} C_VEL
LIN {X 0,Y 199.672,Z 290.425,A -85,B 0,C 180,E1 -21397.221,E2 -21397.221} C_VEL
LIN {X 0,Y 199.748,Z 290.417,A -85,B 0,C 180,E1 -21401.803,E2 -21401.803} C_VEL
LIN {X 0,Y 199.769,Z 290.413,A -85,B 0,C 180,E1 -21405.744,E2 -21405.744} C_VEL
LIN {X 0,Y 200.026,Z 290.365,A -85,B 0,C 180,E1 -21409.882,E2 -21409.882} C_VEL
LIN {X 0,Y 199.997,Z 290.365,A -85,B 0,C 180,E1 -21413.949,E2 -21413.949} C_VEL
LIN {X 0,Y 200.285,Z 290.349,A -85,B 0,C 180,E1 -21417.989,E2 -21417.989} C_VEL
LIN {X 0,Y 200.449,Z 290.322,A -85,B 0,C 180,E1 -21420,E2 -21420} C_VEL
LIN {X 0,Y 199.986,Z 290.357,A -85,B 0,C 180,E1 -21424.031,E2 -21424.031} C_VEL
LIN {X 0,Y 200.073,Z 290.373,A -85,B 0,C 180,E1 -21428.078,E2 -21428.078} C_VEL
LIN {X 0,Y 199.856,Z 290.395,A -85,B 0,C 180,E1 -21432.181,E2 -21432.181} C_VEL
LIN {X 0,Y 199.743,Z 290.395,A -85,B 0,C 180,E1 -21436.349,E2 -21436.349} C_VEL
LIN {X 0,Y 199.644,Z 290.43,A -85,B 0,C 180,E1 -21440.612,E2 -21440.612} C_VEL
LIN {X 0,Y 199.623,Z 290.432,A -85,B 0,C 180,E1 -21444.991,E2 -21444.991} C_VEL
LIN {X 0,Y 199.61,Z 290.431,A -85,B 0,C 180,E1 -21449.533,E2 -21449.533} C_VEL
LIN {X 0,Y 199.668,Z 290.419,A -85,B 0,C 180,E1 -21452.352,E2 -21452.352} C_VEL
LIN {X 0,Y 199.618,Z 290.423,A -85,B 0,C 180,E1 -21456.765,E2 -21456.765} C_VEL
LIN {X 0,Y 199.596,Z 290.436,A -85,B 0,C 180,E1 -21459.331,E2 -21459.331} C_VEL
LIN {X 0,Y 199.566,Z 290.425,A -85,B 0,C 180,E1 -21462.306,E2 -21462.306} C_VEL
LIN {X 0,Y 199.578,Z 290.439,A -85,B 0,C 180,E1 -21465.227,E2 -21465.227} C_VEL
LIN {X 0,Y 199.572,Z 290.432,A -85,B 0,C 180,E1 -21468.002,E2 -21468.002} C_VEL
LIN {X 0,Y 199.599,Z 290.394,A -85,B 0,C 180,E1 -21470.772,E2 -21470.772} C_VEL
